// TIA Portal project "NeuroPLC_S7_1500_DB" (V21)

(* hardware
DEVICE "PLC_1"  S7-1500 station
   slot 0: "导轨_0"  Rack  6ES7 590-1***0-0AA0
   slot 1: "PLC_1"  CPU 1513-1 PN  6ES7 513-1AM03-0AB0  V3.0
      slot 3: "CPU 显示_1"  6ES7591-1AA00-0AA0
      slot 32768: "PROFINET 接口_1"  X1
         slot 32769: "端口_1"  X1 P1
         slot 32770: "端口_2"  X1 P2
      slot 34817: "Virtual CP interface port_1"  Virtual CP interface port  Virtual CP interface port
*)

// ===== PLC "PLC_1"  CPU 1513-1 PN =====

DATA_BLOCK "NeuroPLC_KAN_Weights"   // DB1
{ S7_Optimized_Access := 'TRUE' }
VERSION : 0.1
   VAR
      g0 : Array[0..49] of Real;   // LUT grid (50 pts)
      t1 : Array[0..22399] of Real;   // LUT table (16x28x50)
      w2 : Array[0..447] of Real;   // W(16x28)
      b3 : Array[0..15] of Real;   // bias(16)
      g4 : Array[0..49] of Real;   // LUT grid (50 pts)
      t5 : Array[0..3199] of Real;   // LUT table (4x16x50)
      w6 : Array[0..63] of Real;   // W(4x16)
      b7 : Array[0..3] of Real;   // bias(4)
   END_VAR
BEGIN
   g0[0] := -3.0;
   g0[1] := -2.877551;
   g0[2] := -2.755102;
   g0[3] := -2.632653;
   g0[4] := -2.510204;
   g0[5] := -2.387755;
   g0[6] := -2.265306;
   g0[7] := -2.142857;
   g0[8] := -2.020408;
   g0[9] := -1.897959;
   g0[10] := -1.77551;
   g0[11] := -1.653061;
   g0[12] := -1.530612;
   g0[13] := -1.408163;
   g0[14] := -1.285714;
   g0[15] := -1.163265;
   g0[16] := -1.040816;
   g0[17] := -0.9183673;
   g0[18] := -0.7959184;
   g0[19] := -0.6734694;
   g0[20] := -0.5510204;
   g0[21] := -0.4285714;
   g0[22] := -0.3061224;
   g0[23] := -0.1836735;
   g0[24] := -0.0612245;
   g0[25] := 0.0612245;
   g0[26] := 0.1836735;
   g0[27] := 0.3061224;
   g0[28] := 0.4285714;
   g0[29] := 0.5510204;
   g0[30] := 0.6734694;
   g0[31] := 0.7959184;
   g0[32] := 0.9183673;
   g0[33] := 1.040816;
   g0[34] := 1.163265;
   g0[35] := 1.285714;
   g0[36] := 1.408163;
   g0[37] := 1.530612;
   g0[38] := 1.653061;
   g0[39] := 1.77551;
   g0[40] := 1.897959;
   g0[41] := 2.020408;
   g0[42] := 2.142857;
   g0[43] := 2.265306;
   g0[44] := 2.387755;
   g0[45] := 2.510204;
   g0[46] := 2.632653;
   g0[47] := 2.755102;
   g0[48] := 2.877551;
   g0[49] := 3.0;
   t1[0] := -0.1194829;
   t1[1] := -0.122035;
   t1[2] := -0.1242069;
   t1[3] := -0.1259919;
   t1[4] := -0.1273833;
   t1[5] := -0.1283744;
   t1[6] := -0.1289582;
   t1[7] := -0.1291282;
   t1[8] := -0.1288773;
   t1[9] := -0.1281951;
   t1[10] := -0.1270687;
   t1[11] := -0.125485;
   t1[12] := -0.1234307;
   t1[13] := -0.120893;
   t1[14] := -0.1178586;
   t1[15] := -0.1143145;
   t1[16] := -0.1102476;
   t1[17] := -0.1056448;
   t1[18] := -0.100493;
   t1[19] := -0.0947791;
   t1[20] := -0.0884901;
   t1[21] := -0.0816128;
   t1[22] := -0.0741341;
   t1[23] := -0.066041;
   t1[24] := -0.0573203;
   t1[25] := -0.047959;
   t1[26] := -0.037944;
   t1[27] := -0.0272626;
   t1[28] := -0.0159457;
   t1[29] := -0.0041073;
   t1[30] := 0.0081295;
   t1[31] := 0.0206416;
   t1[32] := 0.033306;
   t1[33] := 0.0459995;
   t1[34] := 0.0585989;
   t1[35] := 0.0709812;
   t1[36] := 0.0830233;
   t1[37] := 0.094602;
   t1[38] := 0.1055942;
   t1[39] := 0.1158768;
   t1[40] := 0.1253268;
   t1[41] := 0.1338208;
   t1[42] := 0.141236;
   t1[43] := 0.1474491;
   t1[44] := 0.1523371;
   t1[45] := 0.1557767;
   t1[46] := 0.157645;
   t1[47] := 0.157853;
   t1[48] := 0.1564832;
   t1[49] := 0.1536715;
   t1[50] := -0.0048413;
   t1[51] := -0.005683;
   t1[52] := -0.0062711;
   t1[53] := -0.0065729;
   t1[54] := -0.0065558;
   t1[55] := -0.0061871;
   t1[56] := -0.0054341;
   t1[57] := -0.0042641;
   t1[58] := -0.0026466;
   t1[59] := -0.000584;
   t1[60] := 0.0018956;
   t1[61] := 0.0047632;
   t1[62] := 0.0079898;
   t1[63] := 0.0115464;
   t1[64] := 0.0154041;
   t1[65] := 0.0195339;
   t1[66] := 0.023907;
   t1[67] := 0.0284943;
   t1[68] := 0.0332668;
   t1[69] := 0.0381957;
   t1[70] := 0.043252;
   t1[71] := 0.0484067;
   t1[72] := 0.0536308;
   t1[73] := 0.0588955;
   t1[74] := 0.0641717;
   t1[75] := 0.0694305;
   t1[76] := 0.074643;
   t1[77] := 0.0797802;
   t1[78] := 0.0848193;
   t1[79] := 0.0897488;
   t1[80] := 0.0945588;
   t1[81] := 0.0992389;
   t1[82] := 0.1037792;
   t1[83] := 0.1081694;
   t1[84] := 0.1123995;
   t1[85] := 0.1164593;
   t1[86] := 0.1203387;
   t1[87] := 0.1240276;
   t1[88] := 0.1275157;
   t1[89] := 0.1307932;
   t1[90] := 0.1338497;
   t1[91] := 0.1366751;
   t1[92] := 0.1392594;
   t1[93] := 0.1415924;
   t1[94] := 0.143664;
   t1[95] := 0.145464;
   t1[96] := 0.1469824;
   t1[97] := 0.148212;
   t1[98] := 0.1491608;
   t1[99] := 0.1498416;
   t1[100] := -0.08693;
   t1[101] := -0.0868943;
   t1[102] := -0.0860951;
   t1[103] := -0.0844797;
   t1[104] := -0.0819952;
   t1[105] := -0.0785887;
   t1[106] := -0.0742075;
   t1[107] := -0.0687987;
   t1[108] := -0.062315;
   t1[109] := -0.054794;
   t1[110] := -0.0463402;
   t1[111] := -0.0370597;
   t1[112] := -0.027059;
   t1[113] := -0.0164442;
   t1[114] := -0.0053218;
   t1[115] := 0.0062022;
   t1[116] := 0.0180213;
   t1[117] := 0.0300293;
   t1[118] := 0.0421199;
   t1[119] := 0.0541869;
   t1[120] := 0.0661239;
   t1[121] := 0.0778248;
   t1[122] := 0.0891831;
   t1[123] := 0.1000927;
   t1[124] := 0.1104472;
   t1[125] := 0.1201404;
   t1[126] := 0.1290659;
   t1[127] := 0.137118;
   t1[128] := 0.144237;
   t1[129] := 0.1504508;
   t1[130] := 0.1557971;
   t1[131] := 0.1603135;
   t1[132] := 0.164038;
   t1[133] := 0.167008;
   t1[134] := 0.1692614;
   t1[135] := 0.1708359;
   t1[136] := 0.1717691;
   t1[137] := 0.1720988;
   t1[138] := 0.1718626;
   t1[139] := 0.1710983;
   t1[140] := 0.1698437;
   t1[141] := 0.1681363;
   t1[142] := 0.166014;
   t1[143] := 0.1635143;
   t1[144] := 0.1606752;
   t1[145] := 0.1575341;
   t1[146] := 0.1541289;
   t1[147] := 0.1504959;
   t1[148] := 0.1466652;
   t1[149] := 0.1426646;
   t1[150] := -0.0762567;
   t1[151] := -0.0788049;
   t1[152] := -0.0811656;
   t1[153] := -0.0833268;
   t1[154] := -0.0852762;
   t1[155] := -0.0870019;
   t1[156] := -0.0884917;
   t1[157] := -0.0897336;
   t1[158] := -0.0907153;
   t1[159] := -0.0914228;
   t1[160] := -0.0918409;
   t1[161] := -0.0919541;
   t1[162] := -0.0917472;
   t1[163] := -0.0912047;
   t1[164] := -0.0903113;
   t1[165] := -0.0890516;
   t1[166] := -0.0874103;
   t1[167] := -0.0853719;
   t1[168] := -0.0829212;
   t1[169] := -0.0800428;
   t1[170] := -0.0767213;
   t1[171] := -0.0729412;
   t1[172] := -0.0686874;
   t1[173] := -0.0639444;
   t1[174] := -0.0586968;
   t1[175] := -0.0529293;
   t1[176] := -0.0466265;
   t1[177] := -0.0397733;
   t1[178] := -0.0323818;
   t1[179] := -0.0245156;
   t1[180] := -0.0162441;
   t1[181] := -0.0076365;
   t1[182] := 0.0012375;
   t1[183] := 0.0103088;
   t1[184] := 0.0195079;
   t1[185] := 0.0287655;
   t1[186] := 0.0380121;
   t1[187] := 0.0471784;
   t1[188] := 0.0561951;
   t1[189] := 0.0649926;
   t1[190] := 0.0735018;
   t1[191] := 0.081653;
   t1[192] := 0.0893772;
   t1[193] := 0.0966047;
   t1[194] := 0.1032663;
   t1[195] := 0.1092926;
   t1[196] := 0.1146141;
   t1[197] := 0.1191739;
   t1[198] := 0.1229757;
   t1[199] := 0.1260427;
   t1[200] := -0.1835549;
   t1[201] := -0.1875302;
   t1[202] := -0.1909346;
   t1[203] := -0.1937087;
   t1[204] := -0.1957933;
   t1[205] := -0.1971291;
   t1[206] := -0.1976567;
   t1[207] := -0.1973169;
   t1[208] := -0.1960545;
   t1[209] := -0.1938767;
   t1[210] := -0.1908398;
   t1[211] := -0.1870016;
   t1[212] := -0.1824198;
   t1[213] := -0.1771521;
   t1[214] := -0.1712564;
   t1[215] := -0.1647903;
   t1[216] := -0.1578115;
   t1[217] := -0.1503778;
   t1[218] := -0.1425468;
   t1[219] := -0.1343765;
   t1[220] := -0.1259243;
   t1[221] := -0.1172482;
   t1[222] := -0.1084058;
   t1[223] := -0.0994548;
   t1[224] := -0.090453;
   t1[225] := -0.0814582;
   t1[226] := -0.072528;
   t1[227] := -0.0637199;
   t1[228] := -0.055075;
   t1[229] := -0.0466024;
   t1[230] := -0.0383076;
   t1[231] := -0.0301963;
   t1[232] := -0.0222742;
   t1[233] := -0.0145468;
   t1[234] := -0.0070199;
   t1[235] := 0.000301;
   t1[236] := 0.0074102;
   t1[237] := 0.0143022;
   t1[238] := 0.0209712;
   t1[239] := 0.0274116;
   t1[240] := 0.0336179;
   t1[241] := 0.0395843;
   t1[242] := 0.0453052;
   t1[243] := 0.0507751;
   t1[244] := 0.0559883;
   t1[245] := 0.0609391;
   t1[246] := 0.0656219;
   t1[247] := 0.0700293;
   t1[248] := 0.0741443;
   t1[249] := 0.077947;
   t1[250] := -0.0558672;
   t1[251] := -0.0568254;
   t1[252] := -0.0574402;
   t1[253] := -0.0577113;
   t1[254] := -0.0576384;
   t1[255] := -0.0572213;
   t1[256] := -0.0564598;
   t1[257] := -0.0553535;
   t1[258] := -0.0539027;
   t1[259] := -0.0521149;
   t1[260] := -0.0500035;
   t1[261] := -0.0475818;
   t1[262] := -0.0448633;
   t1[263] := -0.0418615;
   t1[264] := -0.0385897;
   t1[265] := -0.0350615;
   t1[266] := -0.0312902;
   t1[267] := -0.0272894;
   t1[268] := -0.0230723;
   t1[269] := -0.0186526;
   t1[270] := -0.0140436;
   t1[271] := -0.0092587;
   t1[272] := -0.0043115;
   t1[273] := 0.0007848;
   t1[274] := 0.0060165;
   t1[275] := 0.0113703;
   t1[276] := 0.0168327;
   t1[277] := 0.0223902;
   t1[278] := 0.02802;
   t1[279] := 0.0336815;
   t1[280] := 0.0393322;
   t1[281] := 0.0449295;
   t1[282] := 0.0504309;
   t1[283] := 0.0557939;
   t1[284] := 0.0609759;
   t1[285] := 0.0659345;
   t1[286] := 0.0706271;
   t1[287] := 0.0750112;
   t1[288] := 0.0790442;
   t1[289] := 0.0826836;
   t1[290] := 0.0858869;
   t1[291] := 0.0886116;
   t1[292] := 0.0908151;
   t1[293] := 0.0924549;
   t1[294] := 0.0934885;
   t1[295] := 0.0938734;
   t1[296] := 0.0935669;
   t1[297] := 0.0925394;
   t1[298] := 0.0908244;
   t1[299] := 0.0884755;
   t1[300] := 0.1269326;
   t1[301] := 0.1321426;
   t1[302] := 0.1371375;
   t1[303] := 0.1418623;
   t1[304] := 0.1462617;
   t1[305] := 0.1502807;
   t1[306] := 0.153864;
   t1[307] := 0.1569568;
   t1[308] := 0.1595052;
   t1[309] := 0.1614799;
   t1[310] := 0.1628701;
   t1[311] := 0.1636658;
   t1[312] := 0.1638568;
   t1[313] := 0.1634329;
   t1[314] := 0.1623842;
   t1[315] := 0.1607004;
   t1[316] := 0.1583713;
   t1[317] := 0.155387;
   t1[318] := 0.1517373;
   t1[319] := 0.1474119;
   t1[320] := 0.142401;
   t1[321] := 0.1366941;
   t1[322] := 0.1302814;
   t1[323] := 0.1231525;
   t1[324] := 0.1152975;
   t1[325] := 0.1067062;
   t1[326] := 0.0973684;
   t1[327] := 0.0872743;
   t1[328] := 0.0764416;
   t1[329] := 0.0649405;
   t1[330] := 0.0528468;
   t1[331] := 0.0402367;
   t1[332] := 0.0271859;
   t1[333] := 0.0137705;
   t1[334] := 6.64E-05;
   t1[335] := -0.0138503;
   t1[336] := -0.0279039;
   t1[337] := -0.0420182;
   t1[338] := -0.0561173;
   t1[339] := -0.0701254;
   t1[340] := -0.0839663;
   t1[341] := -0.0975642;
   t1[342] := -0.1108431;
   t1[343] := -0.123727;
   t1[344] := -0.1361401;
   t1[345] := -0.1480062;
   t1[346] := -0.1592495;
   t1[347] := -0.1698008;
   t1[348] := -0.1796257;
   t1[349] := -0.1887;
   t1[350] := -0.0070284;
   t1[351] := -0.0172373;
   t1[352] := -0.0269702;
   t1[353] := -0.0361019;
   t1[354] := -0.0445073;
   t1[355] := -0.0520614;
   t1[356] := -0.058639;
   t1[357] := -0.064115;
   t1[358] := -0.0683716;
   t1[359] := -0.0714012;
   t1[360] := -0.0732835;
   t1[361] := -0.0741003;
   t1[362] := -0.0739335;
   t1[363] := -0.0728651;
   t1[364] := -0.0709769;
   t1[365] := -0.0683507;
   t1[366] := -0.0650686;
   t1[367] := -0.0612124;
   t1[368] := -0.056864;
   t1[369] := -0.0521053;
   t1[370] := -0.0470183;
   t1[371] := -0.0416847;
   t1[372] := -0.0361865;
   t1[373] := -0.0306056;
   t1[374] := -0.0250239;
   t1[375] := -0.0195233;
   t1[376] := -0.0141857;
   t1[377] := -0.0090927;
   t1[378] := -0.0042989;
   t1[379] := 0.0001924;
   t1[380] := 0.0043839;
   t1[381] := 0.0082781;
   t1[382] := 0.0118774;
   t1[383] := 0.0151844;
   t1[384] := 0.0182018;
   t1[385] := 0.0209318;
   t1[386] := 0.0233773;
   t1[387] := 0.0255405;
   t1[388] := 0.0274242;
   t1[389] := 0.0290307;
   t1[390] := 0.0303627;
   t1[391] := 0.0314227;
   t1[392] := 0.0322132;
   t1[393] := 0.0327368;
   t1[394] := 0.0329959;
   t1[395] := 0.0329931;
   t1[396] := 0.032731;
   t1[397] := 0.0322134;
   t1[398] := 0.0314506;
   t1[399] := 0.0304549;
   t1[400] := -0.1028974;
   t1[401] := -0.1051299;
   t1[402] := -0.106706;
   t1[403] := -0.1075951;
   t1[404] := -0.1077664;
   t1[405] := -0.1071893;
   t1[406] := -0.1058333;
   t1[407] := -0.1036677;
   t1[408] := -0.1006654;
   t1[409] := -0.0968557;
   t1[410] := -0.0923118;
   t1[411] := -0.0871083;
   t1[412] := -0.0813197;
   t1[413] := -0.0750206;
   t1[414] := -0.0682854;
   t1[415] := -0.0611888;
   t1[416] := -0.0538051;
   t1[417] := -0.0462091;
   t1[418] := -0.0384752;
   t1[419] := -0.0306779;
   t1[420] := -0.0228918;
   t1[421] := -0.0151914;
   t1[422] := -0.0076512;
   t1[423] := -0.0003457;
   t1[424] := 0.0066504;
   t1[425] := 0.0132627;
   t1[426] := 0.0194167;
   t1[427] := 0.0250381;
   t1[428] := 0.030083;
   t1[429] := 0.0345653;
   t1[430] := 0.0385055;
   t1[431] := 0.0419237;
   t1[432] := 0.0448404;
   t1[433] := 0.0472758;
   t1[434] := 0.0492503;
   t1[435] := 0.0507842;
   t1[436] := 0.0518979;
   t1[437] := 0.0526116;
   t1[438] := 0.0529456;
   t1[439] := 0.0529204;
   t1[440] := 0.0525563;
   t1[441] := 0.0518735;
   t1[442] := 0.0508923;
   t1[443] := 0.0496332;
   t1[444] := 0.0481165;
   t1[445] := 0.0463624;
   t1[446] := 0.0443913;
   t1[447] := 0.0422223;
   t1[448] := 0.0398682;
   t1[449] := 0.0373401;
   t1[450] := 0.0462424;
   t1[451] := 0.039385;
   t1[452] := 0.0330871;
   t1[453] := 0.0274556;
   t1[454] := 0.0225975;
   t1[455] := 0.0186195;
   t1[456] := 0.0156288;
   t1[457] := 0.0137322;
   t1[458] := 0.0130303;
   t1[459] := 0.0135263;
   t1[460] := 0.0151465;
   t1[461] := 0.017815;
   t1[462] := 0.0214562;
   t1[463] := 0.0259943;
   t1[464] := 0.0313536;
   t1[465] := 0.0374582;
   t1[466] := 0.0442325;
   t1[467] := 0.0516006;
   t1[468] := 0.0594868;
   t1[469] := 0.0678154;
   t1[470] := 0.0765106;
   t1[471] := 0.0854967;
   t1[472] := 0.0946978;
   t1[473] := 0.1040383;
   t1[474] := 0.1134424;
   t1[475] := 0.1228343;
   t1[476] := 0.1321382;
   t1[477] := 0.1412786;
   t1[478] := 0.1501878;
   t1[479] := 0.1588135;
   t1[480] := 0.1671054;
   t1[481] := 0.1750129;
   t1[482] := 0.1824855;
   t1[483] := 0.1894727;
   t1[484] := 0.1959241;
   t1[485] := 0.2017891;
   t1[486] := 0.2070173;
   t1[487] := 0.2115581;
   t1[488] := 0.2153611;
   t1[489] := 0.2183758;
   t1[490] := 0.2205516;
   t1[491] := 0.2218381;
   t1[492] := 0.2221848;
   t1[493] := 0.2215413;
   t1[494] := 0.2198569;
   t1[495] := 0.2170812;
   t1[496] := 0.2131638;
   t1[497] := 0.2080761;
   t1[498] := 0.2018998;
   t1[499] := 0.1947507;
   t1[500] := 0.2054697;
   t1[501] := 0.1990182;
   t1[502] := 0.191913;
   t1[503] := 0.1842029;
   t1[504] := 0.1759365;
   t1[505] := 0.1671624;
   t1[506] := 0.1579293;
   t1[507] := 0.1482858;
   t1[508] := 0.1382816;
   t1[509] := 0.1279794;
   t1[510] := 0.1174526;
   t1[511] := 0.1067746;
   t1[512] := 0.0960191;
   t1[513] := 0.0852596;
   t1[514] := 0.0745698;
   t1[515] := 0.0640231;
   t1[516] := 0.0536932;
   t1[517] := 0.0436537;
   t1[518] := 0.0339781;
   t1[519] := 0.02474;
   t1[520] := 0.016013;
   t1[521] := 0.0078706;
   t1[522] := 0.0003865;
   t1[523] := -0.0063659;
   t1[524] := -0.0123129;
   t1[525] := -0.0173809;
   t1[526] := -0.0214963;
   t1[527] := -0.0245862;
   t1[528] := -0.0266352;
   t1[529] := -0.0277371;
   t1[530] := -0.0279982;
   t1[531] := -0.0275248;
   t1[532] := -0.0264229;
   t1[533] := -0.0247989;
   t1[534] := -0.0227588;
   t1[535] := -0.0204089;
   t1[536] := -0.0178554;
   t1[537] := -0.0152045;
   t1[538] := -0.0125623;
   t1[539] := -0.0100351;
   t1[540] := -0.007729;
   t1[541] := -0.0057503;
   t1[542] := -0.0042051;
   t1[543] := -0.0031996;
   t1[544] := -0.0028401;
   t1[545] := -0.0032327;
   t1[546] := -0.0044836;
   t1[547] := -0.0066716;
   t1[548] := -0.0097388;
   t1[549] := -0.0135843;
   t1[550] := 0.069604;
   t1[551] := 0.0578812;
   t1[552] := 0.0457085;
   t1[553] := 0.0331352;
   t1[554] := 0.0202103;
   t1[555] := 0.0069832;
   t1[556] := -0.0064972;
   t1[557] := -0.0201817;
   t1[558] := -0.0340195;
   t1[559] := -0.0479365;
   t1[560] := -0.0618403;
   t1[561] := -0.0756379;
   t1[562] := -0.0892361;
   t1[563] := -0.1025421;
   t1[564] := -0.1154626;
   t1[565] := -0.1279048;
   t1[566] := -0.1397757;
   t1[567] := -0.150982;
   t1[568] := -0.1614309;
   t1[569] := -0.1710294;
   t1[570] := -0.1796844;
   t1[571] := -0.1873028;
   t1[572] := -0.1937916;
   t1[573] := -0.1990579;
   t1[574] := -0.2030086;
   t1[575] := -0.2055506;
   t1[576] := -0.206591;
   t1[577] := -0.2060374;
   t1[578] := -0.2038705;
   t1[579] := -0.2002095;
   t1[580] := -0.1951893;
   t1[581] := -0.1889444;
   t1[582] := -0.1816098;
   t1[583] := -0.1733201;
   t1[584] := -0.16421;
   t1[585] := -0.1544143;
   t1[586] := -0.1440678;
   t1[587] := -0.1333052;
   t1[588] := -0.1222612;
   t1[589] := -0.1110705;
   t1[590] := -0.099868;
   t1[591] := -0.0887883;
   t1[592] := -0.0779662;
   t1[593] := -0.0675364;
   t1[594] := -0.0576337;
   t1[595] := -0.0483928;
   t1[596] := -0.0399484;
   t1[597] := -0.0324114;
   t1[598] := -0.0257726;
   t1[599] := -0.0199858;
   t1[600] := 0.2695681;
   t1[601] := 0.2547651;
   t1[602] := 0.2396336;
   t1[603] := 0.2242566;
   t1[604] := 0.2087173;
   t1[605] := 0.1930988;
   t1[606] := 0.177484;
   t1[607] := 0.1619561;
   t1[608] := 0.1465959;
   t1[609] := 0.1314468;
   t1[610] := 0.1165232;
   t1[611] := 0.1018386;
   t1[612] := 0.0874066;
   t1[613] := 0.0732407;
   t1[614] := 0.0593546;
   t1[615] := 0.0457617;
   t1[616] := 0.0324755;
   t1[617] := 0.0195098;
   t1[618] := 0.0068779;
   t1[619] := -0.0054066;
   t1[620] := -0.01733;
   t1[621] := -0.0288789;
   t1[622] := -0.0400397;
   t1[623] := -0.0507988;
   t1[624] := -0.0611428;
   t1[625] := -0.071058;
   t1[626] := -0.0805309;
   t1[627] := -0.089548;
   t1[628] := -0.0981051;
   t1[629] := -0.1062154;
   t1[630] := -0.1138943;
   t1[631] := -0.1211568;
   t1[632] := -0.1280182;
   t1[633] := -0.1344937;
   t1[634] := -0.1405986;
   t1[635] := -0.146348;
   t1[636] := -0.1517571;
   t1[637] := -0.1568412;
   t1[638] := -0.1616155;
   t1[639] := -0.1660953;
   t1[640] := -0.1702956;
   t1[641] := -0.1742317;
   t1[642] := -0.177919;
   t1[643] := -0.1813724;
   t1[644] := -0.1846074;
   t1[645] := -0.187639;
   t1[646] := -0.1904826;
   t1[647] := -0.1931482;
   t1[648] := -0.1956202;
   t1[649] := -0.1978753;
   t1[650] := 0.1005199;
   t1[651] := 0.1010927;
   t1[652] := 0.1019494;
   t1[653] := 0.1031047;
   t1[654] := 0.1045734;
   t1[655] := 0.1063704;
   t1[656] := 0.1085104;
   t1[657] := 0.1110083;
   t1[658] := 0.1138772;
   t1[659] := 0.1171066;
   t1[660] := 0.1206669;
   t1[661] := 0.1245281;
   t1[662] := 0.1286602;
   t1[663] := 0.1330331;
   t1[664] := 0.1376169;
   t1[665] := 0.1423814;
   t1[666] := 0.1472968;
   t1[667] := 0.1523329;
   t1[668] := 0.1574598;
   t1[669] := 0.1626474;
   t1[670] := 0.1678657;
   t1[671] := 0.1730847;
   t1[672] := 0.1782744;
   t1[673] := 0.1834047;
   t1[674] := 0.1884457;
   t1[675] := 0.1933672;
   t1[676] := 0.1981394;
   t1[677] := 0.2027322;
   t1[678] := 0.2071245;
   t1[679] := 0.2113114;
   t1[680] := 0.2152903;
   t1[681] := 0.2190582;
   t1[682] := 0.2226123;
   t1[683] := 0.2259496;
   t1[684] := 0.2290675;
   t1[685] := 0.231963;
   t1[686] := 0.2346332;
   t1[687] := 0.2370754;
   t1[688] := 0.2392866;
   t1[689] := 0.241264;
   t1[690] := 0.2430048;
   t1[691] := 0.2445061;
   t1[692] := 0.2457651;
   t1[693] := 0.2467789;
   t1[694] := 0.2475446;
   t1[695] := 0.2480595;
   t1[696] := 0.2483206;
   t1[697] := 0.2483248;
   t1[698] := 0.2480676;
   t1[699] := 0.247544;
   t1[700] := 0.0554956;
   t1[701] := 0.0394485;
   t1[702] := 0.0236316;
   t1[703] := 0.008216;
   t1[704] := -0.0066272;
   t1[705] := -0.0207266;
   t1[706] := -0.0339111;
   t1[707] := -0.0460094;
   t1[708] := -0.0568595;
   t1[709] := -0.0664407;
   t1[710] := -0.0748439;
   t1[711] := -0.0821628;
   t1[712] := -0.0884911;
   t1[713] := -0.0939227;
   t1[714] := -0.0985512;
   t1[715] := -0.1024704;
   t1[716] := -0.1057741;
   t1[717] := -0.108556;
   t1[718] := -0.1109099;
   t1[719] := -0.1129296;
   t1[720] := -0.1147089;
   t1[721] := -0.1163414;
   t1[722] := -0.1179209;
   t1[723] := -0.1195412;
   t1[724] := -0.1212961;
   t1[725] := -0.1232793;
   t1[726] := -0.1255845;
   t1[727] := -0.1283051;
   t1[728] := -0.1314804;
   t1[729] := -0.1350474;
   t1[730] := -0.1389318;
   t1[731] := -0.1430591;
   t1[732] := -0.1473549;
   t1[733] := -0.151745;
   t1[734] := -0.1561548;
   t1[735] := -0.1605101;
   t1[736] := -0.1647365;
   t1[737] := -0.1687595;
   t1[738] := -0.1725048;
   t1[739] := -0.175898;
   t1[740] := -0.1788648;
   t1[741] := -0.1813307;
   t1[742] := -0.1832213;
   t1[743] := -0.1844624;
   t1[744] := -0.1849795;
   t1[745] := -0.1846982;
   t1[746] := -0.1835442;
   t1[747] := -0.1814626;
   t1[748] := -0.178497;
   t1[749] := -0.1747214;
   t1[750] := -0.0316489;
   t1[751] := -0.0336773;
   t1[752] := -0.0356129;
   t1[753] := -0.0374797;
   t1[754] := -0.0393015;
   t1[755] := -0.0411025;
   t1[756] := -0.0429063;
   t1[757] := -0.0447371;
   t1[758] := -0.0466166;
   t1[759] := -0.0485351;
   t1[760] := -0.0504581;
   t1[761] := -0.0523502;
   t1[762] := -0.0541761;
   t1[763] := -0.0559007;
   t1[764] := -0.0574886;
   t1[765] := -0.0589045;
   t1[766] := -0.0601133;
   t1[767] := -0.0610795;
   t1[768] := -0.0617679;
   t1[769] := -0.0621433;
   t1[770] := -0.0621704;
   t1[771] := -0.0618138;
   t1[772] := -0.0610385;
   t1[773] := -0.0598089;
   t1[774] := -0.0580899;
   t1[775] := -0.0558463;
   t1[776] := -0.0530426;
   t1[777] := -0.0496441;
   t1[778] := -0.045655;
   t1[779] := -0.041154;
   t1[780] := -0.0362282;
   t1[781] := -0.0309646;
   t1[782] := -0.0254501;
   t1[783] := -0.0197719;
   t1[784] := -0.014017;
   t1[785] := -0.0082723;
   t1[786] := -0.0026249;
   t1[787] := 0.0028383;
   t1[788] := 0.00803;
   t1[789] := 0.0128635;
   t1[790] := 0.0172515;
   t1[791] := 0.0211072;
   t1[792] := 0.0243434;
   t1[793] := 0.0268733;
   t1[794] := 0.0286097;
   t1[795] := 0.0294656;
   t1[796] := 0.029354;
   t1[797] := 0.0282124;
   t1[798] := 0.0261014;
   t1[799] := 0.0231194;
   t1[800] := -0.0541978;
   t1[801] := -0.0467753;
   t1[802] := -0.0388649;
   t1[803] := -0.0305291;
   t1[804] := -0.0218303;
   t1[805] := -0.0128309;
   t1[806] := -0.0035936;
   t1[807] := 0.0058194;
   t1[808] := 0.0153467;
   t1[809] := 0.0249448;
   t1[810] := 0.0345843;
   t1[811] := 0.0442363;
   t1[812] := 0.0538718;
   t1[813] := 0.0634616;
   t1[814] := 0.0729769;
   t1[815] := 0.0823886;
   t1[816] := 0.0916676;
   t1[817] := 0.1007851;
   t1[818] := 0.1097119;
   t1[819] := 0.118419;
   t1[820] := 0.1268776;
   t1[821] := 0.1350584;
   t1[822] := 0.1429326;
   t1[823] := 0.1504711;
   t1[824] := 0.1576449;
   t1[825] := 0.164425;
   t1[826] := 0.1707824;
   t1[827] := 0.1766881;
   t1[828] := 0.1821203;
   t1[829] := 0.1870701;
   t1[830] := 0.1915307;
   t1[831] := 0.1954946;
   t1[832] := 0.1989548;
   t1[833] := 0.2019042;
   t1[834] := 0.2043355;
   t1[835] := 0.2062417;
   t1[836] := 0.2076155;
   t1[837] := 0.2084498;
   t1[838] := 0.2087374;
   t1[839] := 0.2084712;
   t1[840] := 0.2076441;
   t1[841] := 0.2062487;
   t1[842] := 0.2042782;
   t1[843] := 0.2017251;
   t1[844] := 0.1985825;
   t1[845] := 0.1948431;
   t1[846] := 0.1904997;
   t1[847] := 0.1855553;
   t1[848] := 0.1800624;
   t1[849] := 0.1740892;
   t1[850] := 0.0165106;
   t1[851] := 0.0131955;
   t1[852] := 0.0096175;
   t1[853] := 0.0058087;
   t1[854] := 0.0018013;
   t1[855] := -0.0023724;
   t1[856] := -0.0066803;
   t1[857] := -0.0110902;
   t1[858] := -0.0155693;
   t1[859] := -0.020078;
   t1[860] := -0.0245705;
   t1[861] := -0.0290012;
   t1[862] := -0.0333244;
   t1[863] := -0.0374945;
   t1[864] := -0.0414656;
   t1[865] := -0.0451922;
   t1[866] := -0.0486286;
   t1[867] := -0.051729;
   t1[868] := -0.0544477;
   t1[869] := -0.0567391;
   t1[870] := -0.0585574;
   t1[871] := -0.059857;
   t1[872] := -0.0605922;
   t1[873] := -0.0607173;
   t1[874] := -0.0601865;
   t1[875] := -0.0589543;
   t1[876] := -0.0569748;
   t1[877] := -0.0542027;
   t1[878] := -0.050625;
   t1[879] := -0.0462901;
   t1[880] := -0.0412532;
   t1[881] := -0.0355697;
   t1[882] := -0.0292946;
   t1[883] := -0.0224833;
   t1[884] := -0.0151911;
   t1[885] := -0.0074732;
   t1[886] := 0.0006152;
   t1[887] := 0.0090187;
   t1[888] := 0.0176823;
   t1[889] := 0.0265505;
   t1[890] := 0.0355681;
   t1[891] := 0.0446799;
   t1[892] := 0.0538307;
   t1[893] := 0.0629652;
   t1[894] := 0.072028;
   t1[895] := 0.0809641;
   t1[896] := 0.089718;
   t1[897] := 0.0982373;
   t1[898] := 0.1064823;
   t1[899] := 0.1144174;
   t1[900] := 0.2570028;
   t1[901] := 0.2452174;
   t1[902] := 0.2328795;
   t1[903] := 0.2200509;
   t1[904] := 0.2067933;
   t1[905] := 0.1931687;
   t1[906] := 0.1792386;
   t1[907] := 0.1650651;
   t1[908] := 0.150709;
   t1[909] := 0.1362187;
   t1[910] := 0.1216325;
   t1[911] := 0.1069886;
   t1[912] := 0.0923249;
   t1[913] := 0.0776796;
   t1[914] := 0.0630908;
   t1[915] := 0.0485965;
   t1[916] := 0.0342347;
   t1[917] := 0.0200437;
   t1[918] := 0.0060615;
   t1[919] := -0.0076739;
   t1[920] := -0.0211244;
   t1[921] := -0.0342518;
   t1[922] := -0.0470182;
   t1[923] := -0.0593854;
   t1[924] := -0.0713153;
   t1[925] := -0.0827699;
   t1[926] := -0.0937111;
   t1[927] := -0.1041009;
   t1[928] := -0.1139093;
   t1[929] := -0.1231216;
   t1[930] := -0.131725;
   t1[931] := -0.1397063;
   t1[932] := -0.1470526;
   t1[933] := -0.1537509;
   t1[934] := -0.1597883;
   t1[935] := -0.1651517;
   t1[936] := -0.1698283;
   t1[937] := -0.1738049;
   t1[938] := -0.1770687;
   t1[939] := -0.1796066;
   t1[940] := -0.1814057;
   t1[941] := -0.182453;
   t1[942] := -0.1827355;
   t1[943] := -0.1822402;
   t1[944] := -0.1809543;
   t1[945] := -0.1788645;
   t1[946] := -0.1759581;
   t1[947] := -0.172232;
   t1[948] := -0.1677332;
   t1[949] := -0.1625242;
   t1[950] := 0.1695031;
   t1[951] := 0.1635204;
   t1[952] := 0.1571902;
   t1[953] := 0.1505017;
   t1[954] := 0.1434443;
   t1[955] := 0.1360076;
   t1[956] := 0.1281809;
   t1[957] := 0.1199536;
   t1[958] := 0.1113172;
   t1[959] := 0.1022939;
   t1[960] := 0.0929304;
   t1[961] := 0.0832739;
   t1[962] := 0.0733716;
   t1[963] := 0.063271;
   t1[964] := 0.0530191;
   t1[965] := 0.0426633;
   t1[966] := 0.0322509;
   t1[967] := 0.021829;
   t1[968] := 0.0114451;
   t1[969] := 0.0011463;
   t1[970] := -0.0090201;
   t1[971] := -0.0190068;
   t1[972] := -0.0287666;
   t1[973] := -0.0382521;
   t1[974] := -0.0474162;
   t1[975] := -0.0562116;
   t1[976] := -0.0645909;
   t1[977] := -0.0725072;
   t1[978] := -0.0799368;
   t1[979] := -0.0869006;
   t1[980] := -0.0934244;
   t1[981] := -0.099534;
   t1[982] := -0.1052553;
   t1[983] := -0.1106141;
   t1[984] := -0.1156361;
   t1[985] := -0.1203473;
   t1[986] := -0.1247734;
   t1[987] := -0.1289402;
   t1[988] := -0.1328736;
   t1[989] := -0.1365994;
   t1[990] := -0.1401433;
   t1[991] := -0.1435313;
   t1[992] := -0.1467892;
   t1[993] := -0.1499427;
   t1[994] := -0.1530177;
   t1[995] := -0.1560401;
   t1[996] := -0.1590355;
   t1[997] := -0.1620217;
   t1[998] := -0.164975;
   t1[999] := -0.1678591;
   t1[1000] := -0.189392;
   t1[1001] := -0.1768052;
   t1[1002] := -0.1641579;
   t1[1003] := -0.1515508;
   t1[1004] := -0.1390849;
   t1[1005] := -0.1268609;
   t1[1006] := -0.1149796;
   t1[1007] := -0.1035419;
   t1[1008] := -0.092643;
   t1[1009] := -0.0822929;
   t1[1010] := -0.0724342;
   t1[1011] := -0.0630079;
   t1[1012] := -0.0539548;
   t1[1013] := -0.0452158;
   t1[1014] := -0.0367318;
   t1[1015] := -0.0284437;
   t1[1016] := -0.0202924;
   t1[1017] := -0.0122187;
   t1[1018] := -0.0041636;
   t1[1019] := 0.0039321;
   t1[1020] := 0.0121275;
   t1[1021] := 0.0204816;
   t1[1022] := 0.0290537;
   t1[1023] := 0.0379028;
   t1[1024] := 0.047088;
   t1[1025] := 0.0566685;
   t1[1026] := 0.0667034;
   t1[1027] := 0.0772513;
   t1[1028] := 0.0883329;
   t1[1029] := 0.0998958;
   t1[1030] := 0.1118798;
   t1[1031] := 0.1242244;
   t1[1032] := 0.1368694;
   t1[1033] := 0.1497545;
   t1[1034] := 0.1628193;
   t1[1035] := 0.1760034;
   t1[1036] := 0.1892465;
   t1[1037] := 0.2024884;
   t1[1038] := 0.2156686;
   t1[1039] := 0.2287269;
   t1[1040] := 0.2416029;
   t1[1041] := 0.2542362;
   t1[1042] := 0.2665667;
   t1[1043] := 0.2785338;
   t1[1044] := 0.2900774;
   t1[1045] := 0.301137;
   t1[1046] := 0.3116523;
   t1[1047] := 0.321566;
   t1[1048] := 0.3308358;
   t1[1049] := 0.3394241;
   t1[1050] := -0.0330082;
   t1[1051] := -0.0413051;
   t1[1052] := -0.0491068;
   t1[1053] := -0.0562725;
   t1[1054] := -0.062661;
   t1[1055] := -0.0681315;
   t1[1056] := -0.0725428;
   t1[1057] := -0.0757542;
   t1[1058] := -0.0776326;
   t1[1059] := -0.0781712;
   t1[1060] := -0.0774618;
   t1[1061] := -0.0755992;
   t1[1062] := -0.0726782;
   t1[1063] := -0.0687934;
   t1[1064] := -0.0640394;
   t1[1065] := -0.0585112;
   t1[1066] := -0.0523032;
   t1[1067] := -0.0455102;
   t1[1068] := -0.038227;
   t1[1069] := -0.0305481;
   t1[1070] := -0.0225684;
   t1[1071] := -0.0143825;
   t1[1072] := -0.0060852;
   t1[1073] := 0.002229;
   t1[1074] := 0.0104652;
   t1[1075] := 0.0185288;
   t1[1076] := 0.026325;
   t1[1077] := 0.0337595;
   t1[1078] := 0.0407725;
   t1[1079] := 0.0473696;
   t1[1080] := 0.0535637;
   t1[1081] := 0.059368;
   t1[1082] := 0.0647953;
   t1[1083] := 0.0698586;
   t1[1084] := 0.074571;
   t1[1085] := 0.0789453;
   t1[1086] := 0.0829946;
   t1[1087] := 0.0867319;
   t1[1088] := 0.0901701;
   t1[1089] := 0.0933223;
   t1[1090] := 0.0962013;
   t1[1091] := 0.0988202;
   t1[1092] := 0.101192;
   t1[1093] := 0.1033297;
   t1[1094] := 0.1052462;
   t1[1095] := 0.1069545;
   t1[1096] := 0.1084676;
   t1[1097] := 0.109796;
   t1[1098] := 0.1109382;
   t1[1099] := 0.1118888;
   t1[1100] := -0.0263191;
   t1[1101] := -0.01451;
   t1[1102] := -0.0032086;
   t1[1103] := 0.0074345;
   t1[1104] := 0.0172688;
   t1[1105] := 0.0261435;
   t1[1106] := 0.0339082;
   t1[1107] := 0.0404122;
   t1[1108] := 0.0455144;
   t1[1109] := 0.0492193;
   t1[1110] := 0.0516466;
   t1[1111] := 0.0529186;
   t1[1112] := 0.0531581;
   t1[1113] := 0.0524875;
   t1[1114] := 0.0510294;
   t1[1115] := 0.0489064;
   t1[1116] := 0.046241;
   t1[1117] := 0.0431558;
   t1[1118] := 0.0397734;
   t1[1119] := 0.0362162;
   t1[1120] := 0.0326069;
   t1[1121] := 0.0290681;
   t1[1122] := 0.0257222;
   t1[1123] := 0.0226918;
   t1[1124] := 0.0200995;
   t1[1125] := 0.0180679;
   t1[1126] := 0.0167195;
   t1[1127] := 0.0161764;
   t1[1128] := 0.0165029;
   t1[1129] := 0.0176541;
   t1[1130] := 0.019573;
   t1[1131] := 0.0222024;
   t1[1132] := 0.0254852;
   t1[1133] := 0.0293642;
   t1[1134] := 0.0337824;
   t1[1135] := 0.0386827;
   t1[1136] := 0.0440079;
   t1[1137] := 0.049701;
   t1[1138] := 0.0557048;
   t1[1139] := 0.0619621;
   t1[1140] := 0.068416;
   t1[1141] := 0.0750092;
   t1[1142] := 0.0816847;
   t1[1143] := 0.0883854;
   t1[1144] := 0.0950541;
   t1[1145] := 0.1016337;
   t1[1146] := 0.1080671;
   t1[1147] := 0.1143009;
   t1[1148] := 0.1202996;
   t1[1149] := 0.1260335;
   t1[1150] := 0.0412466;
   t1[1151] := 0.0424801;
   t1[1152] := 0.0432831;
   t1[1153] := 0.0436424;
   t1[1154] := 0.0435449;
   t1[1155] := 0.0429775;
   t1[1156] := 0.041927;
   t1[1157] := 0.0403802;
   t1[1158] := 0.0383267;
   t1[1159] := 0.0357943;
   t1[1160] := 0.0328415;
   t1[1161] := 0.0295276;
   t1[1162] := 0.0259119;
   t1[1163] := 0.0220536;
   t1[1164] := 0.018012;
   t1[1165] := 0.0138463;
   t1[1166] := 0.0096158;
   t1[1167] := 0.0053798;
   t1[1168] := 0.0011976;
   t1[1169] := -0.0028716;
   t1[1170] := -0.0067686;
   t1[1171] := -0.010434;
   t1[1172] := -0.0138085;
   t1[1173] := -0.0168331;
   t1[1174] := -0.0194482;
   t1[1175] := -0.0215948;
   t1[1176] := -0.0232134;
   t1[1177] := -0.0242452;
   t1[1178] := -0.0246632;
   t1[1179] := -0.0245009;
   t1[1180] := -0.0237986;
   t1[1181] := -0.0225969;
   t1[1182] := -0.020936;
   t1[1183] := -0.0188563;
   t1[1184] := -0.0163981;
   t1[1185] := -0.0136019;
   t1[1186] := -0.0105081;
   t1[1187] := -0.0071569;
   t1[1188] := -0.0035887;
   t1[1189] := 0.000156;
   t1[1190] := 0.004037;
   t1[1191] := 0.0080138;
   t1[1192] := 0.0120461;
   t1[1193] := 0.0160935;
   t1[1194] := 0.0201156;
   t1[1195] := 0.0240721;
   t1[1196] := 0.0279227;
   t1[1197] := 0.0316308;
   t1[1198] := 0.0351799;
   t1[1199] := 0.0385597;
   t1[1200] := 0.1668451;
   t1[1201] := 0.157337;
   t1[1202] := 0.1473946;
   t1[1203] := 0.1370998;
   t1[1204] := 0.1265343;
   t1[1205] := 0.1157796;
   t1[1206] := 0.1049176;
   t1[1207] := 0.0940298;
   t1[1208] := 0.0831964;
   t1[1209] := 0.0724736;
   t1[1210] := 0.0618986;
   t1[1211] := 0.0515082;
   t1[1212] := 0.0413391;
   t1[1213] := 0.0314279;
   t1[1214] := 0.0218116;
   t1[1215] := 0.0125267;
   t1[1216] := 0.0036101;
   t1[1217] := -0.0049014;
   t1[1218] := -0.0129713;
   t1[1219] := -0.0205627;
   t1[1220] := -0.0276389;
   t1[1221] := -0.0341632;
   t1[1222] := -0.0400987;
   t1[1223] := -0.0454088;
   t1[1224] := -0.0500568;
   t1[1225] := -0.0540058;
   t1[1226] := -0.0572192;
   t1[1227] := -0.0596604;
   t1[1228] := -0.0613163;
   t1[1229] := -0.0622176;
   t1[1230] := -0.0624005;
   t1[1231] := -0.0619007;
   t1[1232] := -0.0607542;
   t1[1233] := -0.058997;
   t1[1234] := -0.0566648;
   t1[1235] := -0.0537936;
   t1[1236] := -0.0504193;
   t1[1237] := -0.0465778;
   t1[1238] := -0.042305;
   t1[1239] := -0.0376369;
   t1[1240] := -0.0326093;
   t1[1241] := -0.0272581;
   t1[1242] := -0.0216192;
   t1[1243] := -0.0157286;
   t1[1244] := -0.0096221;
   t1[1245] := -0.0033357;
   t1[1246] := 0.0030947;
   t1[1247] := 0.0096327;
   t1[1248] := 0.016239;
   t1[1249] := 0.0228733;
   t1[1250] := -0.2291011;
   t1[1251] := -0.2228987;
   t1[1252] := -0.216103;
   t1[1253] := -0.208726;
   t1[1254] := -0.20078;
   t1[1255] := -0.1922772;
   t1[1256] := -0.1832296;
   t1[1257] := -0.1736495;
   t1[1258] := -0.1635502;
   t1[1259] := -0.1529613;
   t1[1260] := -0.1419253;
   t1[1261] := -0.1304853;
   t1[1262] := -0.1186842;
   t1[1263] := -0.1065649;
   t1[1264] := -0.0941705;
   t1[1265] := -0.0815438;
   t1[1266] := -0.0687279;
   t1[1267] := -0.0557656;
   t1[1268] := -0.0426999;
   t1[1269] := -0.0295739;
   t1[1270] := -0.0164303;
   t1[1271] := -0.0033123;
   t1[1272] := 0.0097374;
   t1[1273] := 0.0226756;
   t1[1274] := 0.0354595;
   t1[1275] := 0.0480461;
   t1[1276] := 0.0603924;
   t1[1277] := 0.0724556;
   t1[1278] := 0.0841977;
   t1[1279] := 0.0955904;
   t1[1280] := 0.1066066;
   t1[1281] := 0.1172188;
   t1[1282] := 0.1273999;
   t1[1283] := 0.1371226;
   t1[1284] := 0.1463595;
   t1[1285] := 0.1550836;
   t1[1286] := 0.1632674;
   t1[1287] := 0.1708837;
   t1[1288] := 0.1779052;
   t1[1289] := 0.1843048;
   t1[1290] := 0.1900551;
   t1[1291] := 0.1951288;
   t1[1292] := 0.1994988;
   t1[1293] := 0.2031377;
   t1[1294] := 0.2060182;
   t1[1295] := 0.2081131;
   t1[1296] := 0.2093952;
   t1[1297] := 0.209847;
   t1[1298] := 0.2095002;
   t1[1299] := 0.2084018;
   t1[1300] := 0.0971736;
   t1[1301] := 0.0893726;
   t1[1302] := 0.0816981;
   t1[1303] := 0.0742237;
   t1[1304] := 0.0670231;
   t1[1305] := 0.0601697;
   t1[1306] := 0.0537372;
   t1[1307] := 0.0477992;
   t1[1308] := 0.0424258;
   t1[1309] := 0.0376323;
   t1[1310] := 0.0333909;
   t1[1311] := 0.0296728;
   t1[1312] := 0.0264492;
   t1[1313] := 0.023691;
   t1[1314] := 0.0213695;
   t1[1315] := 0.0194558;
   t1[1316] := 0.0179209;
   t1[1317] := 0.0167361;
   t1[1318] := 0.0158723;
   t1[1319] := 0.0153008;
   t1[1320] := 0.0149927;
   t1[1321] := 0.014919;
   t1[1322] := 0.0150509;
   t1[1323] := 0.0153595;
   t1[1324] := 0.015816;
   t1[1325] := 0.0163914;
   t1[1326] := 0.0170568;
   t1[1327] := 0.0177835;
   t1[1328] := 0.0185539;
   t1[1329] := 0.0193714;
   t1[1330] := 0.0202419;
   t1[1331] := 0.0211712;
   t1[1332] := 0.0221653;
   t1[1333] := 0.0232299;
   t1[1334] := 0.0243709;
   t1[1335] := 0.0255942;
   t1[1336] := 0.0269056;
   t1[1337] := 0.028311;
   t1[1338] := 0.0298162;
   t1[1339] := 0.0314271;
   t1[1340] := 0.0331496;
   t1[1341] := 0.0349894;
   t1[1342] := 0.0369525;
   t1[1343] := 0.0390447;
   t1[1344] := 0.0412719;
   t1[1345] := 0.0436399;
   t1[1346] := 0.0461545;
   t1[1347] := 0.0488163;
   t1[1348] := 0.0515983;
   t1[1349] := 0.0544655;
   t1[1350] := 0.1530943;
   t1[1351] := 0.1526932;
   t1[1352] := 0.151513;
   t1[1353] := 0.1494604;
   t1[1354] := 0.1464418;
   t1[1355] := 0.1423638;
   t1[1356] := 0.1371326;
   t1[1357] := 0.1306549;
   t1[1358] := 0.1228458;
   t1[1359] := 0.1137522;
   t1[1360] := 0.103525;
   t1[1361] := 0.0923181;
   t1[1362] := 0.0802852;
   t1[1363] := 0.0675802;
   t1[1364] := 0.0543566;
   t1[1365] := 0.0407684;
   t1[1366] := 0.0269692;
   t1[1367] := 0.013113;
   t1[1368] := -0.0006467;
   t1[1369] := -0.014156;
   t1[1370] := -0.0272612;
   t1[1371] := -0.0398084;
   t1[1372] := -0.051644;
   t1[1373] := -0.0626141;
   t1[1374] := -0.0725651;
   t1[1375] := -0.081343;
   t1[1376] := -0.0887943;
   t1[1377] := -0.0947657;
   t1[1378] := -0.0991863;
   t1[1379] := -0.1021403;
   t1[1380] := -0.1037292;
   t1[1381] := -0.1040546;
   t1[1382] := -0.1032181;
   t1[1383] := -0.1013212;
   t1[1384] := -0.0984656;
   t1[1385] := -0.0947527;
   t1[1386] := -0.0902843;
   t1[1387] := -0.0851617;
   t1[1388] := -0.0794867;
   t1[1389] := -0.0733608;
   t1[1390] := -0.0668855;
   t1[1391] := -0.0601624;
   t1[1392] := -0.0532932;
   t1[1393] := -0.0463793;
   t1[1394] := -0.0395223;
   t1[1395] := -0.0328239;
   t1[1396] := -0.0263856;
   t1[1397] := -0.0202947;
   t1[1398] := -0.0145677;
   t1[1399] := -0.0091988;
   t1[1400] := -0.1092411;
   t1[1401] := -0.1088026;
   t1[1402] := -0.107988;
   t1[1403] := -0.1067583;
   t1[1404] := -0.1050746;
   t1[1405] := -0.1028977;
   t1[1406] := -0.1001886;
   t1[1407] := -0.0969084;
   t1[1408] := -0.0930205;
   t1[1409] := -0.0885262;
   t1[1410] := -0.0834569;
   t1[1411] := -0.0778447;
   t1[1412] := -0.0717218;
   t1[1413] := -0.0651204;
   t1[1414] := -0.0580724;
   t1[1415] := -0.0506102;
   t1[1416] := -0.0427658;
   t1[1417] := -0.0345714;
   t1[1418] := -0.0260591;
   t1[1419] := -0.017261;
   t1[1420] := -0.0082092;
   t1[1421] := 0.0010639;
   t1[1422] := 0.0105265;
   t1[1423] := 0.0201462;
   t1[1424] := 0.0298911;
   t1[1425] := 0.0397288;
   t1[1426] := 0.0496274;
   t1[1427] := 0.0595547;
   t1[1428] := 0.0694891;
   t1[1429] := 0.0794287;
   t1[1430] := 0.0893739;
   t1[1431] := 0.0993248;
   t1[1432] := 0.109282;
   t1[1433] := 0.1192455;
   t1[1434] := 0.1292159;
   t1[1435] := 0.1391932;
   t1[1436] := 0.1491779;
   t1[1437] := 0.1591703;
   t1[1438] := 0.1691706;
   t1[1439] := 0.1791793;
   t1[1440] := 0.1891965;
   t1[1441] := 0.1992225;
   t1[1442] := 0.2092578;
   t1[1443] := 0.2193026;
   t1[1444] := 0.2293572;
   t1[1445] := 0.2394219;
   t1[1446] := 0.249497;
   t1[1447] := 0.2595751;
   t1[1448] := 0.2696103;
   t1[1449] := 0.2795447;
   t1[1450] := -0.1311382;
   t1[1451] := -0.1293386;
   t1[1452] := -0.1270692;
   t1[1453] := -0.1243363;
   t1[1454] := -0.1211458;
   t1[1455] := -0.1175041;
   t1[1456] := -0.1134172;
   t1[1457] := -0.1088914;
   t1[1458] := -0.1039331;
   t1[1459] := -0.0985572;
   t1[1460] := -0.0927844;
   t1[1461] := -0.0866358;
   t1[1462] := -0.0801324;
   t1[1463] := -0.0732953;
   t1[1464] := -0.0661454;
   t1[1465] := -0.0587038;
   t1[1466] := -0.0509916;
   t1[1467] := -0.0430297;
   t1[1468] := -0.0348392;
   t1[1469] := -0.0264412;
   t1[1470] := -0.0178567;
   t1[1471] := -0.0091066;
   t1[1472] := -0.0002121;
   t1[1473] := 0.0088059;
   t1[1474] := 0.0179262;
   t1[1475] := 0.0271279;
   t1[1476] := 0.03639;
   t1[1477] := 0.0456913;
   t1[1478] := 0.0550137;
   t1[1479] := 0.0643438;
   t1[1480] := 0.073669;
   t1[1481] := 0.0829765;
   t1[1482] := 0.0922537;
   t1[1483] := 0.1014878;
   t1[1484] := 0.1106663;
   t1[1485] := 0.1197764;
   t1[1486] := 0.1288054;
   t1[1487] := 0.1377407;
   t1[1488] := 0.1465695;
   t1[1489] := 0.1552792;
   t1[1490] := 0.163857;
   t1[1491] := 0.1722903;
   t1[1492] := 0.1805664;
   t1[1493] := 0.1886727;
   t1[1494] := 0.1965963;
   t1[1495] := 0.2043247;
   t1[1496] := 0.2118451;
   t1[1497] := 0.2191418;
   t1[1498] := 0.2261835;
   t1[1499] := 0.232934;
   t1[1500] := -0.2517078;
   t1[1501] := -0.255779;
   t1[1502] := -0.2592178;
   t1[1503] := -0.2619836;
   t1[1504] := -0.2640356;
   t1[1505] := -0.2653331;
   t1[1506] := -0.2658352;
   t1[1507] := -0.2655013;
   t1[1508] := -0.2642928;
   t1[1509] := -0.2622057;
   t1[1510] := -0.2592635;
   t1[1511] := -0.2554899;
   t1[1512] := -0.2509092;
   t1[1513] := -0.2455452;
   t1[1514] := -0.2394219;
   t1[1515] := -0.2325635;
   t1[1516] := -0.2249937;
   t1[1517] := -0.2167368;
   t1[1518] := -0.2078166;
   t1[1519] := -0.1982572;
   t1[1520] := -0.1880826;
   t1[1521] := -0.1773168;
   t1[1522] := -0.1659838;
   t1[1523] := -0.1541075;
   t1[1524] := -0.141712;
   t1[1525] := -0.1288214;
   t1[1526] := -0.1154595;
   t1[1527] := -0.1016505;
   t1[1528] := -0.0874226;
   t1[1529] := -0.0728122;
   t1[1530] := -0.0578567;
   t1[1531] := -0.0425932;
   t1[1532] := -0.0270591;
   t1[1533] := -0.0112917;
   t1[1534] := 0.0046719;
   t1[1535] := 0.0207941;
   t1[1536] := 0.0370379;
   t1[1537] := 0.0533659;
   t1[1538] := 0.0697409;
   t1[1539] := 0.0861255;
   t1[1540] := 0.1024824;
   t1[1541] := 0.1187744;
   t1[1542] := 0.1349643;
   t1[1543] := 0.1510147;
   t1[1544] := 0.1668883;
   t1[1545] := 0.1825478;
   t1[1546] := 0.197956;
   t1[1547] := 0.2130717;
   t1[1548] := 0.2278336;
   t1[1549] := 0.2421744;
   t1[1550] := 0.0492069;
   t1[1551] := 0.0473487;
   t1[1552] := 0.0448848;
   t1[1553] := 0.0417536;
   t1[1554] := 0.0378936;
   t1[1555] := 0.0332431;
   t1[1556] := 0.0277405;
   t1[1557] := 0.0213245;
   t1[1558] := 0.0139391;
   t1[1559] := 0.005619;
   t1[1560] := -0.0035302;
   t1[1561] := -0.013401;
   t1[1562] := -0.023886;
   t1[1563] := -0.0348776;
   t1[1564] := -0.0462682;
   t1[1565] := -0.0579503;
   t1[1566] := -0.0698166;
   t1[1567] := -0.0817592;
   t1[1568] := -0.0936709;
   t1[1569] := -0.1054441;
   t1[1570] := -0.1169712;
   t1[1571] := -0.1281447;
   t1[1572] := -0.1388571;
   t1[1573] := -0.149001;
   t1[1574] := -0.1584687;
   t1[1575] := -0.1671527;
   t1[1576] := -0.1749456;
   t1[1577] := -0.1817403;
   t1[1578] := -0.187479;
   t1[1579] := -0.1921975;
   t1[1580] := -0.1959424;
   t1[1581] := -0.1987597;
   t1[1582] := -0.2006959;
   t1[1583] := -0.2017973;
   t1[1584] := -0.2021101;
   t1[1585] := -0.2016807;
   t1[1586] := -0.2005555;
   t1[1587] := -0.1987807;
   t1[1588] := -0.1964026;
   t1[1589] := -0.1934676;
   t1[1590] := -0.1900219;
   t1[1591] := -0.1861119;
   t1[1592] := -0.181784;
   t1[1593] := -0.1770843;
   t1[1594] := -0.1720593;
   t1[1595] := -0.1667552;
   t1[1596] := -0.1612183;
   t1[1597] := -0.1554927;
   t1[1598] := -0.1496101;
   t1[1599] := -0.1435986;
   t1[1600] := 0.2468299;
   t1[1601] := 0.2540316;
   t1[1602] := 0.2604414;
   t1[1603] := 0.2659326;
   t1[1604] := 0.2703789;
   t1[1605] := 0.2736538;
   t1[1606] := 0.2756305;
   t1[1607] := 0.2761828;
   t1[1608] := 0.2751915;
   t1[1609] := 0.2726526;
   t1[1610] := 0.2686527;
   t1[1611] := 0.2632808;
   t1[1612] := 0.2566258;
   t1[1613] := 0.2487768;
   t1[1614] := 0.2398228;
   t1[1615] := 0.2298528;
   t1[1616] := 0.2189557;
   t1[1617] := 0.2072205;
   t1[1618] := 0.1947364;
   t1[1619] := 0.1815922;
   t1[1620] := 0.167877;
   t1[1621] := 0.1536797;
   t1[1622] := 0.1390895;
   t1[1623] := 0.1241952;
   t1[1624] := 0.1090858;
   t1[1625] := 0.0938504;
   t1[1626] := 0.078578;
   t1[1627] := 0.0633574;
   t1[1628] := 0.0482628;
   t1[1629] := 0.0333406;
   t1[1630] := 0.018634;
   t1[1631] := 0.0041861;
   t1[1632] := -0.0099597;
   t1[1633] := -0.0237602;
   t1[1634] := -0.0371722;
   t1[1635] := -0.0501526;
   t1[1636] := -0.0626579;
   t1[1637] := -0.0746451;
   t1[1638] := -0.0860709;
   t1[1639] := -0.096892;
   t1[1640] := -0.1070653;
   t1[1641] := -0.1165475;
   t1[1642] := -0.1252953;
   t1[1643] := -0.1332657;
   t1[1644] := -0.1404152;
   t1[1645] := -0.1467007;
   t1[1646] := -0.152079;
   t1[1647] := -0.1565153;
   t1[1648] := -0.1600175;
   t1[1649] := -0.1626064;
   t1[1650] := -0.0399078;
   t1[1651] := -0.0301289;
   t1[1652] := -0.0201678;
   t1[1653] := -0.0101244;
   t1[1654] := -9.84E-05;
   t1[1655] := 0.0098103;
   t1[1656] := 0.0195017;
   t1[1657] := 0.0288762;
   t1[1658] := 0.0378364;
   t1[1659] := 0.0463278;
   t1[1660] := 0.0543289;
   t1[1661] := 0.0618192;
   t1[1662] := 0.0687783;
   t1[1663] := 0.0751856;
   t1[1664] := 0.0810207;
   t1[1665] := 0.0862631;
   t1[1666] := 0.0908924;
   t1[1667] := 0.0948879;
   t1[1668] := 0.0982293;
   t1[1669] := 0.1008961;
   t1[1670] := 0.1028678;
   t1[1671] := 0.1041238;
   t1[1672] := 0.1046438;
   t1[1673] := 0.1044072;
   t1[1674] := 0.1033935;
   t1[1675] := 0.1015823;
   t1[1676] := 0.0989531;
   t1[1677] := 0.0954857;
   t1[1678] := 0.0911945;
   t1[1679] := 0.0861596;
   t1[1680] := 0.0804685;
   t1[1681] := 0.0742084;
   t1[1682] := 0.0674668;
   t1[1683] := 0.0603311;
   t1[1684] := 0.0528886;
   t1[1685] := 0.0452268;
   t1[1686] := 0.0374331;
   t1[1687] := 0.0295947;
   t1[1688] := 0.0217992;
   t1[1689] := 0.014134;
   t1[1690] := 0.0066863;
   t1[1691] := -0.0004563;
   t1[1692] := -0.0072066;
   t1[1693] := -0.0134771;
   t1[1694] := -0.0191804;
   t1[1695] := -0.0242291;
   t1[1696] := -0.0285359;
   t1[1697] := -0.0320332;
   t1[1698] := -0.0347523;
   t1[1699] := -0.0367556;
   t1[1700] := -0.227583;
   t1[1701] := -0.2247074;
   t1[1702] := -0.2216533;
   t1[1703] := -0.2184904;
   t1[1704] := -0.215288;
   t1[1705] := -0.2121158;
   t1[1706] := -0.2090431;
   t1[1707] := -0.2061395;
   t1[1708] := -0.2034693;
   t1[1709] := -0.201016;
   t1[1710] := -0.1986995;
   t1[1711] := -0.1964381;
   t1[1712] := -0.19415;
   t1[1713] := -0.1917534;
   t1[1714] := -0.1891667;
   t1[1715] := -0.186308;
   t1[1716] := -0.1830956;
   t1[1717] := -0.1794477;
   t1[1718] := -0.1752826;
   t1[1719] := -0.1705185;
   t1[1720] := -0.1650736;
   t1[1721] := -0.1588662;
   t1[1722] := -0.1518145;
   t1[1723] := -0.1438368;
   t1[1724] := -0.1348513;
   t1[1725] := -0.1247762;
   t1[1726] := -0.1135298;
   t1[1727] := -0.1010309;
   t1[1728] := -0.0872722;
   t1[1729] := -0.0723857;
   t1[1730] := -0.056519;
   t1[1731] := -0.0398198;
   t1[1732] := -0.0224358;
   t1[1733] := -0.0045147;
   t1[1734] := 0.013796;
   t1[1735] := 0.0323485;
   t1[1736] := 0.0509951;
   t1[1737] := 0.0695881;
   t1[1738] := 0.08798;
   t1[1739] := 0.1060231;
   t1[1740] := 0.1235696;
   t1[1741] := 0.140472;
   t1[1742] := 0.1565824;
   t1[1743] := 0.1717535;
   t1[1744] := 0.1858373;
   t1[1745] := 0.1986862;
   t1[1746] := 0.2101526;
   t1[1747] := 0.220115;
   t1[1748] := 0.2285822;
   t1[1749] := 0.235604;
   t1[1750] := 0.15399;
   t1[1751] := 0.1538572;
   t1[1752] := 0.1530664;
   t1[1753] := 0.1515775;
   t1[1754] := 0.1493506;
   t1[1755] := 0.1463457;
   t1[1756] := 0.1425229;
   t1[1757] := 0.1378421;
   t1[1758] := 0.1322681;
   t1[1759] := 0.1258384;
   t1[1760] := 0.1186478;
   t1[1761] := 0.1107924;
   t1[1762] := 0.1023686;
   t1[1763] := 0.0934728;
   t1[1764] := 0.084201;
   t1[1765] := 0.0746497;
   t1[1766] := 0.0649152;
   t1[1767] := 0.0550936;
   t1[1768] := 0.0452813;
   t1[1769] := 0.0355746;
   t1[1770] := 0.0260698;
   t1[1771] := 0.0168631;
   t1[1772] := 0.0080508;
   t1[1773] := -0.0002708;
   t1[1774] := -0.0080054;
   t1[1775] := -0.0150567;
   t1[1776] := -0.0213285;
   t1[1777] := -0.0267247;
   t1[1778] := -0.0311856;
   t1[1779] := -0.03472;
   t1[1780] := -0.0373441;
   t1[1781] := -0.0390743;
   t1[1782] := -0.0399271;
   t1[1783] := -0.0399188;
   t1[1784] := -0.0390658;
   t1[1785] := -0.0373845;
   t1[1786] := -0.0348912;
   t1[1787] := -0.0316023;
   t1[1788] := -0.0275342;
   t1[1789] := -0.0227033;
   t1[1790] := -0.017126;
   t1[1791] := -0.0108185;
   t1[1792] := -0.0037974;
   t1[1793] := 0.003921;
   t1[1794] := 0.0123203;
   t1[1795] := 0.0213842;
   t1[1796] := 0.0310963;
   t1[1797] := 0.0414288;
   t1[1798] := 0.0522972;
   t1[1799] := 0.063599;
   t1[1800] := -0.1692545;
   t1[1801] := -0.1719219;
   t1[1802] := -0.1737095;
   t1[1803] := -0.1745087;
   t1[1804] := -0.1742106;
   t1[1805] := -0.1727067;
   t1[1806] := -0.1698882;
   t1[1807] := -0.1656465;
   t1[1808] := -0.1598818;
   t1[1809] := -0.1526316;
   t1[1810] := -0.1440417;
   t1[1811] := -0.1342608;
   t1[1812] := -0.1234376;
   t1[1813] := -0.1117208;
   t1[1814] := -0.099259;
   t1[1815] := -0.086201;
   t1[1816] := -0.0726953;
   t1[1817] := -0.0588908;
   t1[1818] := -0.044936;
   t1[1819] := -0.0309797;
   t1[1820] := -0.0171706;
   t1[1821] := -0.0036572;
   t1[1822] := 0.0094116;
   t1[1823] := 0.0218873;
   t1[1824] := 0.0336211;
   t1[1825] := 0.0444643;
   t1[1826] := 0.0542682;
   t1[1827] := 0.062885;
   t1[1828] := 0.0702438;
   t1[1829] := 0.0764204;
   t1[1830] := 0.0815068;
   t1[1831] := 0.0855952;
   t1[1832] := 0.0887777;
   t1[1833] := 0.0911463;
   t1[1834] := 0.092793;
   t1[1835] := 0.0938102;
   t1[1836] := 0.0942897;
   t1[1837] := 0.0943237;
   t1[1838] := 0.0940042;
   t1[1839] := 0.0934234;
   t1[1840] := 0.0926734;
   t1[1841] := 0.0918462;
   t1[1842] := 0.091034;
   t1[1843] := 0.0903287;
   t1[1844] := 0.0898226;
   t1[1845] := 0.0896076;
   t1[1846] := 0.089776;
   t1[1847] := 0.090402;
   t1[1848] := 0.0914717;
   t1[1849] := 0.0929436;
   t1[1850] := -0.1842585;
   t1[1851] := -0.1840431;
   t1[1852] := -0.1834812;
   t1[1853] := -0.1824941;
   t1[1854] := -0.1810031;
   t1[1855] := -0.1789295;
   t1[1856] := -0.1761944;
   t1[1857] := -0.1727193;
   t1[1858] := -0.1684293;
   t1[1859] := -0.1633116;
   t1[1860] := -0.1574021;
   t1[1861] := -0.1507379;
   t1[1862] := -0.1433562;
   t1[1863] := -0.1352942;
   t1[1864] := -0.126589;
   t1[1865] := -0.1172778;
   t1[1866] := -0.1073979;
   t1[1867] := -0.0969863;
   t1[1868] := -0.0860802;
   t1[1869] := -0.0747169;
   t1[1870] := -0.0629335;
   t1[1871] := -0.050767;
   t1[1872] := -0.0382549;
   t1[1873] := -0.0254341;
   t1[1874] := -0.0123419;
   t1[1875] := 0.0009846;
   t1[1876] := 0.0145081;
   t1[1877] := 0.0281916;
   t1[1878] := 0.0420004;
   t1[1879] := 0.0559045;
   t1[1880] := 0.0698747;
   t1[1881] := 0.0838816;
   t1[1882] := 0.0978958;
   t1[1883] := 0.1118879;
   t1[1884] := 0.1258287;
   t1[1885] := 0.1396887;
   t1[1886] := 0.1534386;
   t1[1887] := 0.167049;
   t1[1888] := 0.1804906;
   t1[1889] := 0.1937339;
   t1[1890] := 0.2067497;
   t1[1891] := 0.2195086;
   t1[1892] := 0.2319812;
   t1[1893] := 0.2441382;
   t1[1894] := 0.2559501;
   t1[1895] := 0.2673877;
   t1[1896] := 0.2784216;
   t1[1897] := 0.2890209;
   t1[1898] := 0.2991468;
   t1[1899] := 0.3087583;
   t1[1900] := -0.3433722;
   t1[1901] := -0.3352931;
   t1[1902] := -0.3264073;
   t1[1903] := -0.3167214;
   t1[1904] := -0.3062419;
   t1[1905] := -0.2949751;
   t1[1906] := -0.2829276;
   t1[1907] := -0.2701057;
   t1[1908] := -0.2565185;
   t1[1909] := -0.2422126;
   t1[1910] := -0.2272647;
   t1[1911] := -0.2117521;
   t1[1912] := -0.1957523;
   t1[1913] := -0.1793427;
   t1[1914] := -0.1626008;
   t1[1915] := -0.1456038;
   t1[1916] := -0.1284292;
   t1[1917] := -0.1111544;
   t1[1918] := -0.0938568;
   t1[1919] := -0.0766139;
   t1[1920] := -0.059503;
   t1[1921] := -0.0426015;
   t1[1922] := -0.0259869;
   t1[1923] := -0.0097365;
   t1[1924] := 0.0060723;
   t1[1925] := 0.021362;
   t1[1926] := 0.0360552;
   t1[1927] := 0.0500748;
   t1[1928] := 0.0633724;
   t1[1929] := 0.0759543;
   t1[1930] := 0.0878328;
   t1[1931] := 0.0990201;
   t1[1932] := 0.1095287;
   t1[1933] := 0.1193707;
   t1[1934] := 0.1285587;
   t1[1935] := 0.1371047;
   t1[1936] := 0.1450212;
   t1[1937] := 0.1523206;
   t1[1938] := 0.159015;
   t1[1939] := 0.1651168;
   t1[1940] := 0.1706384;
   t1[1941] := 0.175592;
   t1[1942] := 0.17999;
   t1[1943] := 0.1838447;
   t1[1944] := 0.1871684;
   t1[1945] := 0.1899734;
   t1[1946] := 0.192272;
   t1[1947] := 0.1940764;
   t1[1948] := 0.1953979;
   t1[1949] := 0.1962473;
   t1[1950] := 0.0363517;
   t1[1951] := 0.0309942;
   t1[1952] := 0.0259224;
   t1[1953] := 0.0212328;
   t1[1954] := 0.0170217;
   t1[1955] := 0.0133855;
   t1[1956] := 0.0104207;
   t1[1957] := 0.0082236;
   t1[1958] := 0.0068848;
   t1[1959] := 0.0064029;
   t1[1960] := 0.0067043;
   t1[1961] := 0.0077135;
   t1[1962] := 0.0093549;
   t1[1963] := 0.0115529;
   t1[1964] := 0.0142321;
   t1[1965] := 0.0173167;
   t1[1966] := 0.0207314;
   t1[1967] := 0.0244004;
   t1[1968] := 0.0282484;
   t1[1969] := 0.0321997;
   t1[1970] := 0.0361787;
   t1[1971] := 0.0401099;
   t1[1972] := 0.0439178;
   t1[1973] := 0.0475268;
   t1[1974] := 0.0508614;
   t1[1975] := 0.0538459;
   t1[1976] := 0.0564049;
   t1[1977] := 0.058463;
   t1[1978] := 0.059982;
   t1[1979] := 0.0609932;
   t1[1980] := 0.0615358;
   t1[1981] := 0.0616491;
   t1[1982] := 0.0613721;
   t1[1983] := 0.0607442;
   t1[1984] := 0.0598046;
   t1[1985] := 0.0585923;
   t1[1986] := 0.0571468;
   t1[1987] := 0.055507;
   t1[1988] := 0.0537123;
   t1[1989] := 0.0518019;
   t1[1990] := 0.0498149;
   t1[1991] := 0.0477906;
   t1[1992] := 0.0457681;
   t1[1993] := 0.0437867;
   t1[1994] := 0.0418856;
   t1[1995] := 0.040104;
   t1[1996] := 0.038481;
   t1[1997] := 0.0370488;
   t1[1998] := 0.0358042;
   t1[1999] := 0.0347328;
   t1[2000] := -0.2135215;
   t1[2001] := -0.1983883;
   t1[2002] := -0.1827447;
   t1[2003] := -0.166669;
   t1[2004] := -0.1502396;
   t1[2005] := -0.1335349;
   t1[2006] := -0.1166332;
   t1[2007] := -0.0996131;
   t1[2008] := -0.0825521;
   t1[2009] := -0.0655172;
   t1[2010] := -0.0485664;
   t1[2011] := -0.0317578;
   t1[2012] := -0.0151492;
   t1[2013] := 0.0012013;
   t1[2014] := 0.0172358;
   t1[2015] := 0.0328962;
   t1[2016] := 0.0481248;
   t1[2017] := 0.0628634;
   t1[2018] := 0.0770541;
   t1[2019] := 0.090639;
   t1[2020] := 0.1035601;
   t1[2021] := 0.1157594;
   t1[2022] := 0.127179;
   t1[2023] := 0.1377609;
   t1[2024] := 0.1474471;
   t1[2025] := 0.1561797;
   t1[2026] := 0.1639007;
   t1[2027] := 0.1705526;
   t1[2028] := 0.1761245;
   t1[2029] := 0.1806938;
   t1[2030] := 0.1843482;
   t1[2031] := 0.1871748;
   t1[2032] := 0.1892613;
   t1[2033] := 0.190695;
   t1[2034] := 0.1915633;
   t1[2035] := 0.1919536;
   t1[2036] := 0.1919534;
   t1[2037] := 0.1916501;
   t1[2038] := 0.1911311;
   t1[2039] := 0.1904838;
   t1[2040] := 0.1897957;
   t1[2041] := 0.1891541;
   t1[2042] := 0.1886465;
   t1[2043] := 0.1883604;
   t1[2044] := 0.188383;
   t1[2045] := 0.1888019;
   t1[2046] := 0.1897045;
   t1[2047] := 0.191155;
   t1[2048] := 0.1931011;
   t1[2049] := 0.1954547;
   t1[2050] := -0.2638247;
   t1[2051] := -0.253926;
   t1[2052] := -0.243357;
   t1[2053] := -0.232141;
   t1[2054] := -0.2203012;
   t1[2055] := -0.2078611;
   t1[2056] := -0.1948439;
   t1[2057] := -0.181273;
   t1[2058] := -0.167174;
   t1[2059] := -0.1526075;
   t1[2060] := -0.1376618;
   t1[2061] := -0.1224262;
   t1[2062] := -0.1069895;
   t1[2063] := -0.0914409;
   t1[2064] := -0.0758695;
   t1[2065] := -0.0603644;
   t1[2066] := -0.0450145;
   t1[2067] := -0.0299091;
   t1[2068] := -0.0151371;
   t1[2069] := -0.0007877;
   t1[2070] := 0.0130502;
   t1[2071] := 0.0262873;
   t1[2072] := 0.0388347;
   t1[2073] := 0.0506033;
   t1[2074] := 0.061504;
   t1[2075] := 0.0714477;
   t1[2076] := 0.0803453;
   t1[2077] := 0.0881083;
   t1[2078] := 0.0947028;
   t1[2079] := 0.1001986;
   t1[2080] := 0.104677;
   t1[2081] := 0.1082193;
   t1[2082] := 0.1109071;
   t1[2083] := 0.1128215;
   t1[2084] := 0.114044;
   t1[2085] := 0.114656;
   t1[2086] := 0.1147388;
   t1[2087] := 0.1143738;
   t1[2088] := 0.1136424;
   t1[2089] := 0.1126258;
   t1[2090] := 0.1114055;
   t1[2091] := 0.1100629;
   t1[2092] := 0.1086792;
   t1[2093] := 0.1073359;
   t1[2094] := 0.1061144;
   t1[2095] := 0.1050959;
   t1[2096] := 0.1043619;
   t1[2097] := 0.1039764;
   t1[2098] := 0.1039163;
   t1[2099] := 0.1041317;
   t1[2100] := -0.0215827;
   t1[2101] := -0.0217664;
   t1[2102] := -0.0220519;
   t1[2103] := -0.0223617;
   t1[2104] := -0.0226185;
   t1[2105] := -0.0227447;
   t1[2106] := -0.0226629;
   t1[2107] := -0.0222959;
   t1[2108] := -0.0215713;
   t1[2109] := -0.0204994;
   t1[2110] := -0.0191547;
   t1[2111] := -0.0176138;
   t1[2112] := -0.015953;
   t1[2113] := -0.0142488;
   t1[2114] := -0.0125777;
   t1[2115] := -0.0110161;
   t1[2116] := -0.0096404;
   t1[2117] := -0.0085271;
   t1[2118] := -0.0077527;
   t1[2119] := -0.0073935;
   t1[2120] := -0.007526;
   t1[2121] := -0.0082266;
   t1[2122] := -0.0095719;
   t1[2123] := -0.0116382;
   t1[2124] := -0.014502;
   t1[2125] := -0.0182397;
   t1[2126] := -0.0229278;
   t1[2127] := -0.0286421;
   t1[2128] := -0.0353979;
   t1[2129] := -0.0430952;
   t1[2130] := -0.0516213;
   t1[2131] := -0.0608633;
   t1[2132] := -0.0707085;
   t1[2133] := -0.081044;
   t1[2134] := -0.0917572;
   t1[2135] := -0.1027351;
   t1[2136] := -0.1138651;
   t1[2137] := -0.1250344;
   t1[2138] := -0.1361301;
   t1[2139] := -0.1470395;
   t1[2140] := -0.1576497;
   t1[2141] := -0.1678481;
   t1[2142] := -0.1775218;
   t1[2143] := -0.1865581;
   t1[2144] := -0.1948441;
   t1[2145] := -0.202267;
   t1[2146] := -0.2087142;
   t1[2147] := -0.2140943;
   t1[2148] := -0.2184236;
   t1[2149] := -0.2217521;
   t1[2150] := 0.0948695;
   t1[2151] := 0.1027036;
   t1[2152] := 0.1098262;
   t1[2153] := 0.116154;
   t1[2154] := 0.1216037;
   t1[2155] := 0.1260919;
   t1[2156] := 0.1295351;
   t1[2157] := 0.1318502;
   t1[2158] := 0.1329586;
   t1[2159] := 0.132856;
   t1[2160] := 0.131597;
   t1[2161] := 0.1292376;
   t1[2162] := 0.1258339;
   t1[2163] := 0.1214417;
   t1[2164] := 0.1161173;
   t1[2165] := 0.1099166;
   t1[2166] := 0.1028956;
   t1[2167] := 0.0951103;
   t1[2168] := 0.0866169;
   t1[2169] := 0.0774713;
   t1[2170] := 0.0677295;
   t1[2171] := 0.0574476;
   t1[2172] := 0.0466816;
   t1[2173] := 0.0354875;
   t1[2174] := 0.0239214;
   t1[2175] := 0.0120393;
   t1[2176] := -0.0001028;
   t1[2177] := -0.0124489;
   t1[2178] := -0.0249446;
   t1[2179] := -0.0375386;
   t1[2180] := -0.05018;
   t1[2181] := -0.0628179;
   t1[2182] := -0.0754015;
   t1[2183] := -0.0878796;
   t1[2184] := -0.1002016;
   t1[2185] := -0.1123164;
   t1[2186] := -0.1241731;
   t1[2187] := -0.1357209;
   t1[2188] := -0.1469087;
   t1[2189] := -0.1576857;
   t1[2190] := -0.168001;
   t1[2191] := -0.1778036;
   t1[2192] := -0.1870427;
   t1[2193] := -0.1956673;
   t1[2194] := -0.2036265;
   t1[2195] := -0.2108694;
   t1[2196] := -0.217345;
   t1[2197] := -0.2230122;
   t1[2198] := -0.2278775;
   t1[2199] := -0.2319627;
   t1[2200] := 0.2239106;
   t1[2201] := 0.2190618;
   t1[2202] := 0.2131876;
   t1[2203] := 0.2063059;
   t1[2204] := 0.1984346;
   t1[2205] := 0.1895914;
   t1[2206] := 0.1797942;
   t1[2207] := 0.1690608;
   t1[2208] := 0.1574113;
   t1[2209] := 0.144899;
   t1[2210] := 0.1316038;
   t1[2211] := 0.1176062;
   t1[2212] := 0.1029866;
   t1[2213] := 0.0878256;
   t1[2214] := 0.0722037;
   t1[2215] := 0.0562014;
   t1[2216] := 0.0398991;
   t1[2217] := 0.0233774;
   t1[2218] := 0.0067168;
   t1[2219] := -0.0100023;
   t1[2220] := -0.0266993;
   t1[2221] := -0.0432937;
   t1[2222] := -0.059705;
   t1[2223] := -0.0758528;
   t1[2224] := -0.0916565;
   t1[2225] := -0.1070356;
   t1[2226] := -0.1219096;
   t1[2227] := -0.1361983;
   t1[2228] := -0.1498503;
   t1[2229] := -0.1628686;
   t1[2230] := -0.1752626;
   t1[2231] := -0.1870415;
   t1[2232] := -0.1982146;
   t1[2233] := -0.208791;
   t1[2234] := -0.2187801;
   t1[2235] := -0.228191;
   t1[2236] := -0.2370331;
   t1[2237] := -0.2453157;
   t1[2238] := -0.2530478;
   t1[2239] := -0.2602389;
   t1[2240] := -0.2668981;
   t1[2241] := -0.2730347;
   t1[2242] := -0.278658;
   t1[2243] := -0.2837772;
   t1[2244] := -0.2884016;
   t1[2245] := -0.2925403;
   t1[2246] := -0.2962027;
   t1[2247] := -0.2993954;
   t1[2248] := -0.3021117;
   t1[2249] := -0.3043406;
   t1[2250] := -0.210152;
   t1[2251] := -0.1990302;
   t1[2252] := -0.1876812;
   t1[2253] := -0.1762033;
   t1[2254] := -0.1646952;
   t1[2255] := -0.153255;
   t1[2256] := -0.1419814;
   t1[2257] := -0.1309727;
   t1[2258] := -0.1203236;
   t1[2259] := -0.1100722;
   t1[2260] := -0.1002113;
   t1[2261] := -0.0907329;
   t1[2262] := -0.0816288;
   t1[2263] := -0.072891;
   t1[2264] := -0.0645113;
   t1[2265] := -0.0564815;
   t1[2266] := -0.0487936;
   t1[2267] := -0.0414393;
   t1[2268] := -0.0344107;
   t1[2269] := -0.0276995;
   t1[2270] := -0.0212975;
   t1[2271] := -0.0151968;
   t1[2272] := -0.0093891;
   t1[2273] := -0.0038663;
   t1[2274] := 0.0013797;
   t1[2275] := 0.006357;
   t1[2276] := 0.0110738;
   t1[2277] := 0.0155381;
   t1[2278] := 0.0197446;
   t1[2279] := 0.0236629;
   t1[2280] := 0.0272598;
   t1[2281] := 0.030502;
   t1[2282] := 0.0333564;
   t1[2283] := 0.0357896;
   t1[2284] := 0.0377684;
   t1[2285] := 0.0392597;
   t1[2286] := 0.0402302;
   t1[2287] := 0.0406466;
   t1[2288] := 0.0404757;
   t1[2289] := 0.0396844;
   t1[2290] := 0.0382393;
   t1[2291] := 0.0361072;
   t1[2292] := 0.0332549;
   t1[2293] := 0.0296492;
   t1[2294] := 0.0252568;
   t1[2295] := 0.0200445;
   t1[2296] := 0.0139791;
   t1[2297] := 0.0070468;
   t1[2298] := -0.000669;
   t1[2299] := -0.0090543;
   t1[2300] := -0.2450845;
   t1[2301] := -0.2353242;
   t1[2302] := -0.2247794;
   t1[2303] := -0.2134059;
   t1[2304] := -0.2011592;
   t1[2305] := -0.1879949;
   t1[2306] := -0.1738686;
   t1[2307] := -0.1587359;
   t1[2308] := -0.1425592;
   t1[2309] := -0.1254039;
   t1[2310] := -0.1074169;
   t1[2311] := -0.0887473;
   t1[2312] := -0.0695441;
   t1[2313] := -0.0499563;
   t1[2314] := -0.0301329;
   t1[2315] := -0.0102231;
   t1[2316] := 0.0096242;
   t1[2317] := 0.0292598;
   t1[2318] := 0.0485348;
   t1[2319] := 0.0673002;
   t1[2320] := 0.0854068;
   t1[2321] := 0.1027057;
   t1[2322] := 0.1190478;
   t1[2323] := 0.134284;
   t1[2324] := 0.1482654;
   t1[2325] := 0.1608428;
   t1[2326] := 0.1718673;
   t1[2327] := 0.1811903;
   t1[2328] := 0.1887307;
   t1[2329] := 0.1945347;
   t1[2330] := 0.1986626;
   t1[2331] := 0.2011748;
   t1[2332] := 0.2021318;
   t1[2333] := 0.201594;
   t1[2334] := 0.1996216;
   t1[2335] := 0.1962753;
   t1[2336] := 0.1916152;
   t1[2337] := 0.185702;
   t1[2338] := 0.1785959;
   t1[2339] := 0.1703573;
   t1[2340] := 0.1610467;
   t1[2341] := 0.1507245;
   t1[2342] := 0.139451;
   t1[2343] := 0.1272867;
   t1[2344] := 0.1142919;
   t1[2345] := 0.1005271;
   t1[2346] := 0.0860527;
   t1[2347] := 0.0709401;
   t1[2348] := 0.0553158;
   t1[2349] := 0.0393236;
   t1[2350] := -0.4248369;
   t1[2351] := -0.4179277;
   t1[2352] := -0.4100263;
   t1[2353] := -0.401115;
   t1[2354] := -0.3911766;
   t1[2355] := -0.3801935;
   t1[2356] := -0.3681482;
   t1[2357] := -0.3550233;
   t1[2358] := -0.3408041;
   t1[2359] := -0.3255194;
   t1[2360] := -0.3092318;
   t1[2361] := -0.2920052;
   t1[2362] := -0.2739031;
   t1[2363] := -0.2549895;
   t1[2364] := -0.235328;
   t1[2365] := -0.2149823;
   t1[2366] := -0.1940161;
   t1[2367] := -0.1724932;
   t1[2368] := -0.1504773;
   t1[2369] := -0.1280321;
   t1[2370] := -0.1052214;
   t1[2371] := -0.0821088;
   t1[2372] := -0.0587582;
   t1[2373] := -0.0352331;
   t1[2374] := -0.0115973;
   t1[2375] := 0.0120853;
   t1[2376] := 0.0357511;
   t1[2377] := 0.0593363;
   t1[2378] := 0.0827594;
   t1[2379] := 0.105906;
   t1[2380] := 0.1286577;
   t1[2381] := 0.1508963;
   t1[2382] := 0.1725036;
   t1[2383] := 0.1933614;
   t1[2384] := 0.2133514;
   t1[2385] := 0.2323554;
   t1[2386] := 0.2502551;
   t1[2387] := 0.2669323;
   t1[2388] := 0.2822687;
   t1[2389] := 0.2961462;
   t1[2390] := 0.3084463;
   t1[2391] := 0.319051;
   t1[2392] := 0.327842;
   t1[2393] := 0.3347012;
   t1[2394] := 0.3395101;
   t1[2395] := 0.3421504;
   t1[2396] := 0.3425042;
   t1[2397] := 0.3404941;
   t1[2398] := 0.3362485;
   t1[2399] := 0.3299596;
   t1[2400] := 0.3017888;
   t1[2401] := 0.2929916;
   t1[2402] := 0.2837368;
   t1[2403] := 0.2740539;
   t1[2404] := 0.2639727;
   t1[2405] := 0.2535227;
   t1[2406] := 0.2427335;
   t1[2407] := 0.2316348;
   t1[2408] := 0.2202557;
   t1[2409] := 0.2086159;
   t1[2410] := 0.196728;
   t1[2411] := 0.1846043;
   t1[2412] := 0.1722573;
   t1[2413] := 0.1596992;
   t1[2414] := 0.1469425;
   t1[2415] := 0.1339995;
   t1[2416] := 0.1208825;
   t1[2417] := 0.1076039;
   t1[2418] := 0.0941761;
   t1[2419] := 0.0806115;
   t1[2420] := 0.0669224;
   t1[2421] := 0.0531211;
   t1[2422] := 0.03922;
   t1[2423] := 0.0252315;
   t1[2424] := 0.011168;
   t1[2425] := -0.0029583;
   t1[2426] := -0.0171348;
   t1[2427] := -0.0313492;
   t1[2428] := -0.0455605;
   t1[2429] := -0.0596748;
   t1[2430] := -0.0735921;
   t1[2431] := -0.0872125;
   t1[2432] := -0.1004361;
   t1[2433] := -0.1131628;
   t1[2434] := -0.1252928;
   t1[2435] := -0.136726;
   t1[2436] := -0.1473625;
   t1[2437] := -0.1571023;
   t1[2438] := -0.1658456;
   t1[2439] := -0.1734923;
   t1[2440] := -0.1799424;
   t1[2441] := -0.1850961;
   t1[2442] := -0.1888533;
   t1[2443] := -0.1911141;
   t1[2444] := -0.1917786;
   t1[2445] := -0.1907468;
   t1[2446] := -0.1879187;
   t1[2447] := -0.1832308;
   t1[2448] := -0.1768013;
   t1[2449] := -0.1688053;
   t1[2450] := 0.2525824;
   t1[2451] := 0.234157;
   t1[2452] := 0.2152379;
   t1[2453] := 0.1959515;
   t1[2454] := 0.1764241;
   t1[2455] := 0.156782;
   t1[2456] := 0.1371515;
   t1[2457] := 0.1176589;
   t1[2458] := 0.0984263;
   t1[2459] := 0.0795105;
   t1[2460] := 0.0609163;
   t1[2461] := 0.0426475;
   t1[2462] := 0.0247079;
   t1[2463] := 0.007101;
   t1[2464] := -0.0101694;
   t1[2465] := -0.0270996;
   t1[2466] := -0.043686;
   t1[2467] := -0.0599248;
   t1[2468] := -0.0758124;
   t1[2469] := -0.0913451;
   t1[2470] := -0.1065192;
   t1[2471] := -0.121331;
   t1[2472] := -0.1357768;
   t1[2473] := -0.1498529;
   t1[2474] := -0.1635557;
   t1[2475] := -0.1768814;
   t1[2476] := -0.1898264;
   t1[2477] := -0.2023869;
   t1[2478] := -0.2145509;
   t1[2479] := -0.2262909;
   t1[2480] := -0.2375775;
   t1[2481] := -0.2483814;
   t1[2482] := -0.2586735;
   t1[2483] := -0.2684242;
   t1[2484] := -0.2776044;
   t1[2485] := -0.2861848;
   t1[2486] := -0.2941359;
   t1[2487] := -0.3014286;
   t1[2488] := -0.3080335;
   t1[2489] := -0.3139214;
   t1[2490] := -0.3190629;
   t1[2491] := -0.3234286;
   t1[2492] := -0.3269894;
   t1[2493] := -0.3297159;
   t1[2494] := -0.3315789;
   t1[2495] := -0.3325488;
   t1[2496] := -0.3325966;
   t1[2497] := -0.3317031;
   t1[2498] := -0.3298996;
   t1[2499] := -0.3272333;
   t1[2500] := 0.1863346;
   t1[2501] := 0.1800162;
   t1[2502] := 0.1729414;
   t1[2503] := 0.1650857;
   t1[2504] := 0.1564246;
   t1[2505] := 0.1469336;
   t1[2506] := 0.1365881;
   t1[2507] := 0.1253638;
   t1[2508] := 0.1132393;
   t1[2509] := 0.1002423;
   t1[2510] := 0.0864392;
   t1[2511] := 0.0718976;
   t1[2512] := 0.0566846;
   t1[2513] := 0.0408679;
   t1[2514] := 0.0245148;
   t1[2515] := 0.0076928;
   t1[2516] := -0.0095309;
   t1[2517] := -0.0270886;
   t1[2518] := -0.044913;
   t1[2519] := -0.0629367;
   t1[2520] := -0.0810922;
   t1[2521] := -0.0993121;
   t1[2522] := -0.1175291;
   t1[2523] := -0.1356757;
   t1[2524] := -0.1536844;
   t1[2525] := -0.1714878;
   t1[2526] := -0.1890186;
   t1[2527] := -0.2062093;
   t1[2528] := -0.2229935;
   t1[2529] := -0.2393069;
   t1[2530] := -0.2550855;
   t1[2531] := -0.2702649;
   t1[2532] := -0.2847811;
   t1[2533] := -0.2985701;
   t1[2534] := -0.3115676;
   t1[2535] := -0.3237095;
   t1[2536] := -0.3349317;
   t1[2537] := -0.3451701;
   t1[2538] := -0.3543605;
   t1[2539] := -0.3624389;
   t1[2540] := -0.369341;
   t1[2541] := -0.3750027;
   t1[2542] := -0.37936;
   t1[2543] := -0.3823487;
   t1[2544] := -0.3839047;
   t1[2545] := -0.3839638;
   t1[2546] := -0.3824619;
   t1[2547] := -0.3793586;
   t1[2548] := -0.3747315;
   t1[2549] := -0.3686952;
   t1[2550] := 0.0815692;
   t1[2551] := 0.0721724;
   t1[2552] := 0.0627858;
   t1[2553] := 0.0534844;
   t1[2554] := 0.0443431;
   t1[2555] := 0.0354371;
   t1[2556] := 0.0268412;
   t1[2557] := 0.0186305;
   t1[2558] := 0.0108776;
   t1[2559] := 0.0036155;
   t1[2560] := -0.0031535;
   t1[2561] := -0.0094281;
   t1[2562] := -0.0152069;
   t1[2563] := -0.0204886;
   t1[2564] := -0.0252718;
   t1[2565] := -0.029555;
   t1[2566] := -0.0333371;
   t1[2567] := -0.0366166;
   t1[2568] := -0.0393921;
   t1[2569] := -0.0416622;
   t1[2570] := -0.0434257;
   t1[2571] := -0.0446811;
   t1[2572] := -0.0454271;
   t1[2573] := -0.0456624;
   t1[2574] := -0.0453855;
   t1[2575] := -0.044595;
   t1[2576] := -0.0432897;
   t1[2577] := -0.0414683;
   t1[2578] := -0.039138;
   t1[2579] := -0.0363222;
   t1[2580] := -0.0330463;
   t1[2581] := -0.0293356;
   t1[2582] := -0.0252153;
   t1[2583] := -0.0207107;
   t1[2584] := -0.0158472;
   t1[2585] := -0.0106499;
   t1[2586] := -0.0051443;
   t1[2587] := 0.0006445;
   t1[2588] := 0.0066911;
   t1[2589] := 0.0129702;
   t1[2590] := 0.0194567;
   t1[2591] := 0.026125;
   t1[2592] := 0.0329501;
   t1[2593] := 0.0399066;
   t1[2594] := 0.0469692;
   t1[2595] := 0.0541127;
   t1[2596] := 0.0613117;
   t1[2597] := 0.0685377;
   t1[2598] := 0.0757459;
   t1[2599] := 0.0828866;
   t1[2600] := 0.0296985;
   t1[2601] := 0.0298958;
   t1[2602] := 0.0298572;
   t1[2603] := 0.0295598;
   t1[2604] := 0.0289804;
   t1[2605] := 0.028096;
   t1[2606] := 0.0268834;
   t1[2607] := 0.0253197;
   t1[2608] := 0.0233825;
   t1[2609] := 0.0210612;
   t1[2610] := 0.0183545;
   t1[2611] := 0.0152612;
   t1[2612] := 0.0117802;
   t1[2613] := 0.0079105;
   t1[2614] := 0.0036509;
   t1[2615] := -0.0009996;
   t1[2616] := -0.0060423;
   t1[2617] := -0.0114781;
   t1[2618] := -0.0173083;
   t1[2619] := -0.0235339;
   t1[2620] := -0.030156;
   t1[2621] := -0.0371757;
   t1[2622] := -0.0445942;
   t1[2623] := -0.0524126;
   t1[2624] := -0.0606318;
   t1[2625] := -0.0692532;
   t1[2626] := -0.0782777;
   t1[2627] := -0.0877063;
   t1[2628] := -0.0975138;
   t1[2629] := -0.1076262;
   t1[2630] := -0.1179638;
   t1[2631] := -0.1284467;
   t1[2632] := -0.1389955;
   t1[2633] := -0.1495303;
   t1[2634] := -0.1599716;
   t1[2635] := -0.1702395;
   t1[2636] := -0.1802546;
   t1[2637] := -0.189937;
   t1[2638] := -0.1992071;
   t1[2639] := -0.2079852;
   t1[2640] := -0.2161917;
   t1[2641] := -0.2237468;
   t1[2642] := -0.230571;
   t1[2643] := -0.2365844;
   t1[2644] := -0.2417075;
   t1[2645] := -0.2458604;
   t1[2646] := -0.2489637;
   t1[2647] := -0.2509559;
   t1[2648] := -0.2518681;
   t1[2649] := -0.2517596;
   t1[2650] := 0.2789594;
   t1[2651] := 0.2709424;
   t1[2652] := 0.2617649;
   t1[2653] := 0.2513233;
   t1[2654] := 0.2395139;
   t1[2655] := 0.2262332;
   t1[2656] := 0.2113774;
   t1[2657] := 0.1948428;
   t1[2658] := 0.1765366;
   t1[2659] := 0.1565279;
   t1[2660] := 0.135014;
   t1[2661] := 0.1121957;
   t1[2662] := 0.0882736;
   t1[2663] := 0.0634485;
   t1[2664] := 0.0379211;
   t1[2665] := 0.0118922;
   t1[2666] := -0.0144376;
   t1[2667] := -0.0408675;
   t1[2668] := -0.0671968;
   t1[2669] := -0.0932248;
   t1[2670] := -0.1187508;
   t1[2671] := -0.1435741;
   t1[2672] := -0.1674938;
   t1[2673] := -0.1903095;
   t1[2674] := -0.2118202;
   t1[2675] := -0.2318252;
   t1[2676] := -0.2501238;
   t1[2677] := -0.2665164;
   t1[2678] := -0.2809054;
   t1[2679] := -0.2933874;
   t1[2680] := -0.304081;
   t1[2681] := -0.3131043;
   t1[2682] := -0.3205758;
   t1[2683] := -0.3266138;
   t1[2684] := -0.3313366;
   t1[2685] := -0.3348626;
   t1[2686] := -0.3373102;
   t1[2687] := -0.3387977;
   t1[2688] := -0.3394434;
   t1[2689] := -0.3393657;
   t1[2690] := -0.3386829;
   t1[2691] := -0.3375134;
   t1[2692] := -0.3359756;
   t1[2693] := -0.3341878;
   t1[2694] := -0.3322684;
   t1[2695] := -0.3303355;
   t1[2696] := -0.3285078;
   t1[2697] := -0.32688;
   t1[2698] := -0.3254305;
   t1[2699] := -0.3241007;
   t1[2700] := -0.0089786;
   t1[2701] := -0.0170903;
   t1[2702] := -0.0249782;
   t1[2703] := -0.0325892;
   t1[2704] := -0.0398705;
   t1[2705] := -0.046769;
   t1[2706] := -0.0532318;
   t1[2707] := -0.0592059;
   t1[2708] := -0.0646412;
   t1[2709] := -0.069531;
   t1[2710] := -0.0739032;
   t1[2711] := -0.0777865;
   t1[2712] := -0.0812096;
   t1[2713] := -0.0842011;
   t1[2714] := -0.0867897;
   t1[2715] := -0.0890041;
   t1[2716] := -0.090873;
   t1[2717] := -0.0924251;
   t1[2718] := -0.0936891;
   t1[2719] := -0.0946936;
   t1[2720] := -0.0954674;
   t1[2721] := -0.0960391;
   t1[2722] := -0.0964375;
   t1[2723] := -0.0966911;
   t1[2724] := -0.0968288;
   t1[2725] := -0.0968791;
   t1[2726] := -0.0968709;
   t1[2727] := -0.0968326;
   t1[2728] := -0.0967854;
   t1[2729] := -0.0967358;
   t1[2730] := -0.096689;
   t1[2731] := -0.09665;
   t1[2732] := -0.0966238;
   t1[2733] := -0.0966156;
   t1[2734] := -0.0966302;
   t1[2735] := -0.0966729;
   t1[2736] := -0.0967486;
   t1[2737] := -0.0968624;
   t1[2738] := -0.0970193;
   t1[2739] := -0.0972244;
   t1[2740] := -0.0974828;
   t1[2741] := -0.0977994;
   t1[2742] := -0.0981794;
   t1[2743] := -0.0986278;
   t1[2744] := -0.0991497;
   t1[2745] := -0.09975;
   t1[2746] := -0.1004339;
   t1[2747] := -0.1012022;
   t1[2748] := -0.1020352;
   t1[2749] := -0.1029065;
   t1[2750] := 0.1839082;
   t1[2751] := 0.1719079;
   t1[2752] := 0.1598567;
   t1[2753] := 0.1477929;
   t1[2754] := 0.1357548;
   t1[2755] := 0.1237808;
   t1[2756] := 0.111909;
   t1[2757] := 0.1001777;
   t1[2758] := 0.0886241;
   t1[2759] := 0.077267;
   t1[2760] := 0.0661109;
   t1[2761] := 0.0551598;
   t1[2762] := 0.0444179;
   t1[2763] := 0.0338891;
   t1[2764] := 0.0235777;
   t1[2765] := 0.0134876;
   t1[2766] := 0.0036229;
   t1[2767] := -0.0060122;
   t1[2768] := -0.0154137;
   t1[2769] := -0.0245775;
   t1[2770] := -0.0334996;
   t1[2771] := -0.0421758;
   t1[2772] := -0.0506021;
   t1[2773] := -0.0587744;
   t1[2774] := -0.0666886;
   t1[2775] := -0.0743406;
   t1[2776] := -0.0817264;
   t1[2777] := -0.088842;
   t1[2778] := -0.0956898;
   t1[2779] := -0.1022846;
   t1[2780] := -0.1086426;
   t1[2781] := -0.1147801;
   t1[2782] := -0.1207133;
   t1[2783] := -0.1264583;
   t1[2784] := -0.1320314;
   t1[2785] := -0.1374487;
   t1[2786] := -0.1427265;
   t1[2787] := -0.1478809;
   t1[2788] := -0.1529282;
   t1[2789] := -0.1578846;
   t1[2790] := -0.1627663;
   t1[2791] := -0.1675894;
   t1[2792] := -0.1723702;
   t1[2793] := -0.1771248;
   t1[2794] := -0.1818696;
   t1[2795] := -0.1866206;
   t1[2796] := -0.1913941;
   t1[2797] := -0.1961968;
   t1[2798] := -0.2009879;
   t1[2799] := -0.2057118;
   t1[2800] := 0.129127;
   t1[2801] := 0.1244142;
   t1[2802] := 0.1193461;
   t1[2803] := 0.1139074;
   t1[2804] := 0.1080832;
   t1[2805] := 0.1018582;
   t1[2806] := 0.0952174;
   t1[2807] := 0.0881457;
   t1[2808] := 0.0806309;
   t1[2809] := 0.0727068;
   t1[2810] := 0.0644431;
   t1[2811] := 0.0559105;
   t1[2812] := 0.0471798;
   t1[2813] := 0.0383219;
   t1[2814] := 0.0294074;
   t1[2815] := 0.0205071;
   t1[2816] := 0.0116917;
   t1[2817] := 0.0030321;
   t1[2818] := -0.0054011;
   t1[2819] := -0.0135371;
   t1[2820] := -0.021305;
   t1[2821] := -0.0286343;
   t1[2822] := -0.035454;
   t1[2823] := -0.0416934;
   t1[2824] := -0.0472819;
   t1[2825] := -0.0521486;
   t1[2826] := -0.0562227;
   t1[2827] := -0.059434;
   t1[2828] := -0.0617627;
   t1[2829] := -0.0632845;
   t1[2830] := -0.0640861;
   t1[2831] := -0.0642538;
   t1[2832] := -0.0638743;
   t1[2833] := -0.0630341;
   t1[2834] := -0.0618197;
   t1[2835] := -0.0603176;
   t1[2836] := -0.0586143;
   t1[2837] := -0.0567965;
   t1[2838] := -0.0549505;
   t1[2839] := -0.053163;
   t1[2840] := -0.0515205;
   t1[2841] := -0.0501094;
   t1[2842] := -0.0490163;
   t1[2843] := -0.0483278;
   t1[2844] := -0.0481303;
   t1[2845] := -0.0485104;
   t1[2846] := -0.0495547;
   t1[2847] := -0.051326;
   t1[2848] := -0.0537697;
   t1[2849] := -0.0567943;
   t1[2850] := 0.1542486;
   t1[2851] := 0.1550493;
   t1[2852] := 0.1557622;
   t1[2853] := 0.1563427;
   t1[2854] := 0.1567464;
   t1[2855] := 0.1569286;
   t1[2856] := 0.1568447;
   t1[2857] := 0.1564502;
   t1[2858] := 0.1557015;
   t1[2859] := 0.15457;
   t1[2860] := 0.1530392;
   t1[2861] := 0.1510926;
   t1[2862] := 0.1487141;
   t1[2863] := 0.1458872;
   t1[2864] := 0.1425956;
   t1[2865] := 0.138823;
   t1[2866] := 0.1345531;
   t1[2867] := 0.1297696;
   t1[2868] := 0.1244561;
   t1[2869] := 0.1185963;
   t1[2870] := 0.1121739;
   t1[2871] := 0.1051726;
   t1[2872] := 0.097576;
   t1[2873] := 0.0893678;
   t1[2874] := 0.0805317;
   t1[2875] := 0.0710514;
   t1[2876] := 0.0609105;
   t1[2877] := 0.0500932;
   t1[2878] := 0.0386272;
   t1[2879] := 0.0266233;
   t1[2880] := 0.0142016;
   t1[2881] := 0.0014821;
   t1[2882] := -0.0114151;
   t1[2883] := -0.02437;
   t1[2884] := -0.0372626;
   t1[2885] := -0.0499728;
   t1[2886] := -0.0623805;
   t1[2887] := -0.0743657;
   t1[2888] := -0.0858084;
   t1[2889] := -0.0965885;
   t1[2890] := -0.106586;
   t1[2891] := -0.1156808;
   t1[2892] := -0.1237528;
   t1[2893] := -0.1306822;
   t1[2894] := -0.1363487;
   t1[2895] := -0.1406323;
   t1[2896] := -0.143413;
   t1[2897] := -0.1445999;
   t1[2898] := -0.1442478;
   t1[2899] := -0.1424568;
   t1[2900] := 0.2432433;
   t1[2901] := 0.2353556;
   t1[2902] := 0.2270421;
   t1[2903] := 0.2183365;
   t1[2904] := 0.209273;
   t1[2905] := 0.1998853;
   t1[2906] := 0.1902075;
   t1[2907] := 0.1802735;
   t1[2908] := 0.1701179;
   t1[2909] := 0.1597853;
   t1[2910] := 0.1493282;
   t1[2911] := 0.1387992;
   t1[2912] := 0.128251;
   t1[2913] := 0.1177363;
   t1[2914] := 0.1073077;
   t1[2915] := 0.097018;
   t1[2916] := 0.0869198;
   t1[2917] := 0.0770657;
   t1[2918] := 0.0675085;
   t1[2919] := 0.0583008;
   t1[2920] := 0.0494953;
   t1[2921] := 0.0411446;
   t1[2922] := 0.0333014;
   t1[2923] := 0.0260185;
   t1[2924] := 0.0193484;
   t1[2925] := 0.0133438;
   t1[2926] := 0.0080575;
   t1[2927] := 0.0035418;
   t1[2928] := -0.0001807;
   t1[2929] := -0.0031441;
   t1[2930] := -0.0053886;
   t1[2931] := -0.0069547;
   t1[2932] := -0.0078826;
   t1[2933] := -0.0082128;
   t1[2934] := -0.0079854;
   t1[2935] := -0.007241;
   t1[2936] := -0.0060198;
   t1[2937] := -0.0043621;
   t1[2938] := -0.0023084;
   t1[2939] := 0.0001011;
   t1[2940] := 0.0028261;
   t1[2941] := 0.0058261;
   t1[2942] := 0.0090608;
   t1[2943] := 0.01249;
   t1[2944] := 0.0160732;
   t1[2945] := 0.0197702;
   t1[2946] := 0.0235405;
   t1[2947] := 0.027347;
   t1[2948] := 0.0311682;
   t1[2949] := 0.0349876;
   t1[2950] := 0.0060134;
   t1[2951] := 0.0075953;
   t1[2952] := 0.0095188;
   t1[2953] := 0.01177;
   t1[2954] := 0.0143348;
   t1[2955] := 0.017199;
   t1[2956] := 0.0203486;
   t1[2957] := 0.0237696;
   t1[2958] := 0.0274472;
   t1[2959] := 0.0313589;
   t1[2960] := 0.0354757;
   t1[2961] := 0.0397684;
   t1[2962] := 0.0442078;
   t1[2963] := 0.0487648;
   t1[2964] := 0.0534102;
   t1[2965] := 0.0581149;
   t1[2966] := 0.0628497;
   t1[2967] := 0.0675854;
   t1[2968] := 0.0722929;
   t1[2969] := 0.076943;
   t1[2970] := 0.0815065;
   t1[2971] := 0.0859543;
   t1[2972] := 0.0902573;
   t1[2973] := 0.0943862;
   t1[2974] := 0.0983119;
   t1[2975] := 0.1020052;
   t1[2976] := 0.105437;
   t1[2977] := 0.1085783;
   t1[2978] := 0.111415;
   t1[2979] := 0.1139619;
   t1[2980] := 0.1162366;
   t1[2981] := 0.118257;
   t1[2982] := 0.1200409;
   t1[2983] := 0.121606;
   t1[2984] := 0.1229703;
   t1[2985] := 0.1241514;
   t1[2986] := 0.1251671;
   t1[2987] := 0.1260353;
   t1[2988] := 0.1267737;
   t1[2989] := 0.1274002;
   t1[2990] := 0.1279325;
   t1[2991] := 0.1283884;
   t1[2992] := 0.1287857;
   t1[2993] := 0.1291423;
   t1[2994] := 0.1294759;
   t1[2995] := 0.1298042;
   t1[2996] := 0.1301452;
   t1[2997] := 0.1305105;
   t1[2998] := 0.1308815;
   t1[2999] := 0.1312302;
   t1[3000] := 0.1256087;
   t1[3001] := 0.1352973;
   t1[3002] := 0.1443325;
   t1[3003] := 0.152559;
   t1[3004] := 0.1598216;
   t1[3005] := 0.165965;
   t1[3006] := 0.170834;
   t1[3007] := 0.1742733;
   t1[3008] := 0.1761368;
   t1[3009] := 0.1764177;
   t1[3010] := 0.1752191;
   t1[3011] := 0.1726473;
   t1[3012] := 0.1688082;
   t1[3013] := 0.163808;
   t1[3014] := 0.1577529;
   t1[3015] := 0.1507489;
   t1[3016] := 0.1429021;
   t1[3017] := 0.1343186;
   t1[3018] := 0.1251047;
   t1[3019] := 0.1153662;
   t1[3020] := 0.1052095;
   t1[3021] := 0.0947405;
   t1[3022] := 0.0840654;
   t1[3023] := 0.0732903;
   t1[3024] := 0.0625214;
   t1[3025] := 0.0518646;
   t1[3026] := 0.0414262;
   t1[3027] := 0.0313121;
   t1[3028] := 0.0216062;
   t1[3029] := 0.0123507;
   t1[3030] := 0.0035835;
   t1[3031] := -0.0046578;
   t1[3032] := -0.0123355;
   t1[3033] := -0.019412;
   t1[3034] := -0.0258496;
   t1[3035] := -0.0316105;
   t1[3036] := -0.0366572;
   t1[3037] := -0.0409519;
   t1[3038] := -0.0444569;
   t1[3039] := -0.0471346;
   t1[3040] := -0.0489473;
   t1[3041] := -0.0498573;
   t1[3042] := -0.049827;
   t1[3043] := -0.0488186;
   t1[3044] := -0.0467944;
   t1[3045] := -0.0437169;
   t1[3046] := -0.0395483;
   t1[3047] := -0.0342693;
   t1[3048] := -0.0279528;
   t1[3049] := -0.0207005;
   t1[3050] := 0.0231812;
   t1[3051] := 0.0164768;
   t1[3052] := 0.0097991;
   t1[3053] := 0.0031845;
   t1[3054] := -0.0033309;
   t1[3055] := -0.009711;
   t1[3056] := -0.0159195;
   t1[3057] := -0.0219202;
   t1[3058] := -0.0276777;
   t1[3059] := -0.0331666;
   t1[3060] := -0.0383697;
   t1[3061] := -0.0432701;
   t1[3062] := -0.0478508;
   t1[3063] := -0.0520948;
   t1[3064] := -0.0559851;
   t1[3065] := -0.0595047;
   t1[3066] := -0.0626367;
   t1[3067] := -0.0653641;
   t1[3068] := -0.0676698;
   t1[3069] := -0.0695369;
   t1[3070] := -0.0709485;
   t1[3071] := -0.0718874;
   t1[3072] := -0.0723369;
   t1[3073] := -0.0722798;
   t1[3074] := -0.0716991;
   t1[3075] := -0.070578;
   t1[3076] := -0.0688994;
   t1[3077] := -0.0666465;
   t1[3078] := -0.0638269;
   t1[3079] := -0.0604939;
   t1[3080] := -0.0567063;
   t1[3081] := -0.0525226;
   t1[3082] := -0.0480013;
   t1[3083] := -0.0432012;
   t1[3084] := -0.0381807;
   t1[3085] := -0.0329986;
   t1[3086] := -0.0277133;
   t1[3087] := -0.0223835;
   t1[3088] := -0.0170678;
   t1[3089] := -0.0118248;
   t1[3090] := -0.0067131;
   t1[3091] := -0.0017912;
   t1[3092] := 0.0028822;
   t1[3093] := 0.0072485;
   t1[3094] := 0.0112491;
   t1[3095] := 0.0148255;
   t1[3096] := 0.017919;
   t1[3097] := 0.020481;
   t1[3098] := 0.022513;
   t1[3099] := 0.0240322;
   t1[3100] := -0.038803;
   t1[3101] := -0.041465;
   t1[3102] := -0.0442218;
   t1[3103] := -0.0471058;
   t1[3104] := -0.050149;
   t1[3105] := -0.0533837;
   t1[3106] := -0.0568421;
   t1[3107] := -0.0605563;
   t1[3108] := -0.0645558;
   t1[3109] := -0.0688262;
   t1[3110] := -0.0733187;
   t1[3111] := -0.0779837;
   t1[3112] := -0.0827715;
   t1[3113] := -0.0876325;
   t1[3114] := -0.0925168;
   t1[3115] := -0.097375;
   t1[3116] := -0.1021573;
   t1[3117] := -0.106814;
   t1[3118] := -0.1112955;
   t1[3119] := -0.115552;
   t1[3120] := -0.119534;
   t1[3121] := -0.1231917;
   t1[3122] := -0.1264755;
   t1[3123] := -0.1293356;
   t1[3124] := -0.1317225;
   t1[3125] := -0.1335863;
   t1[3126] := -0.1348776;
   t1[3127] := -0.1355469;
   t1[3128] := -0.1355845;
   t1[3129] := -0.135056;
   t1[3130] := -0.1340351;
   t1[3131] := -0.1325956;
   t1[3132] := -0.1308115;
   t1[3133] := -0.1287565;
   t1[3134] := -0.1265045;
   t1[3135] := -0.1241293;
   t1[3136] := -0.1217048;
   t1[3137] := -0.1193047;
   t1[3138] := -0.117003;
   t1[3139] := -0.1148734;
   t1[3140] := -0.1129898;
   t1[3141] := -0.111426;
   t1[3142] := -0.1102559;
   t1[3143] := -0.1095533;
   t1[3144] := -0.109392;
   t1[3145] := -0.1098459;
   t1[3146] := -0.1109888;
   t1[3147] := -0.112873;
   t1[3148] := -0.1154429;
   t1[3149] := -0.1186093;
   t1[3150] := 0.0876806;
   t1[3151] := 0.0804098;
   t1[3152] := 0.0733107;
   t1[3153] := 0.0664517;
   t1[3154] := 0.0599012;
   t1[3155] := 0.0537276;
   t1[3156] := 0.0479992;
   t1[3157] := 0.0427845;
   t1[3158] := 0.0381484;
   t1[3159] := 0.0341009;
   t1[3160] := 0.0306092;
   t1[3161] := 0.027639;
   t1[3162] := 0.0251565;
   t1[3163] := 0.0231273;
   t1[3164] := 0.0215176;
   t1[3165] := 0.020293;
   t1[3166] := 0.0194197;
   t1[3167] := 0.0188633;
   t1[3168] := 0.01859;
   t1[3169] := 0.0185655;
   t1[3170] := 0.0187558;
   t1[3171] := 0.0191267;
   t1[3172] := 0.0196442;
   t1[3173] := 0.0202742;
   t1[3174] := 0.0209826;
   t1[3175] := 0.0217353;
   t1[3176] := 0.0224981;
   t1[3177] := 0.0232371;
   t1[3178] := 0.0239225;
   t1[3179] := 0.0245327;
   t1[3180] := 0.0250472;
   t1[3181] := 0.0254454;
   t1[3182] := 0.0257066;
   t1[3183] := 0.0258103;
   t1[3184] := 0.0257358;
   t1[3185] := 0.0254626;
   t1[3186] := 0.0249699;
   t1[3187] := 0.0242373;
   t1[3188] := 0.0232441;
   t1[3189] := 0.0219697;
   t1[3190] := 0.0203935;
   t1[3191] := 0.0184949;
   t1[3192] := 0.0162533;
   t1[3193] := 0.013648;
   t1[3194] := 0.0106585;
   t1[3195] := 0.0072642;
   t1[3196] := 0.0034444;
   t1[3197] := -0.0008121;
   t1[3198] := -0.0054704;
   t1[3199] := -0.0104808;
   t1[3200] := 0.156688;
   t1[3201] := 0.1584898;
   t1[3202] := 0.1597388;
   t1[3203] := 0.1603476;
   t1[3204] := 0.1602288;
   t1[3205] := 0.159295;
   t1[3206] := 0.1574585;
   t1[3207] := 0.154632;
   t1[3208] := 0.1507343;
   t1[3209] := 0.1457798;
   t1[3210] := 0.1398588;
   t1[3211] := 0.1330631;
   t1[3212] := 0.1254851;
   t1[3213] := 0.1172166;
   t1[3214] := 0.1083499;
   t1[3215] := 0.098977;
   t1[3216] := 0.08919;
   t1[3217] := 0.0790811;
   t1[3218] := 0.0687422;
   t1[3219] := 0.0582655;
   t1[3220] := 0.047743;
   t1[3221] := 0.037267;
   t1[3222] := 0.0269294;
   t1[3223] := 0.0168223;
   t1[3224] := 0.0070378;
   t1[3225] := -0.0023319;
   t1[3226] := -0.0111948;
   t1[3227] := -0.0194591;
   t1[3228] := -0.0270664;
   t1[3229] := -0.0340217;
   t1[3230] := -0.0403372;
   t1[3231] := -0.0460248;
   t1[3232] := -0.0510966;
   t1[3233] := -0.0555648;
   t1[3234] := -0.0594414;
   t1[3235] := -0.0627384;
   t1[3236] := -0.0654681;
   t1[3237] := -0.0676423;
   t1[3238] := -0.0692732;
   t1[3239] := -0.0703729;
   t1[3240] := -0.0709534;
   t1[3241] := -0.0710269;
   t1[3242] := -0.0706053;
   t1[3243] := -0.0697009;
   t1[3244] := -0.0683255;
   t1[3245] := -0.0664914;
   t1[3246] := -0.0642106;
   t1[3247] := -0.0614983;
   t1[3248] := -0.0583853;
   t1[3249] := -0.0549072;
   t1[3250] := -0.031862;
   t1[3251] := -0.035804;
   t1[3252] := -0.039725;
   t1[3253] := -0.0436243;
   t1[3254] := -0.0475011;
   t1[3255] := -0.0513548;
   t1[3256] := -0.0551847;
   t1[3257] := -0.05899;
   t1[3258] := -0.0627687;
   t1[3259] := -0.0664977;
   t1[3260] := -0.0701374;
   t1[3261] := -0.0736476;
   t1[3262] := -0.0769884;
   t1[3263] := -0.0801197;
   t1[3264] := -0.0830013;
   t1[3265] := -0.0855932;
   t1[3266] := -0.0878554;
   t1[3267] := -0.0897477;
   t1[3268] := -0.0912301;
   t1[3269] := -0.0922625;
   t1[3270] := -0.0928049;
   t1[3271] := -0.0928171;
   t1[3272] := -0.0922591;
   t1[3273] := -0.0910909;
   t1[3274] := -0.0892723;
   t1[3275] := -0.0867632;
   t1[3276] := -0.0835237;
   t1[3277] := -0.0795138;
   t1[3278] := -0.0747269;
   t1[3279] := -0.0692185;
   t1[3280] := -0.063051;
   t1[3281] := -0.0562872;
   t1[3282] := -0.0489895;
   t1[3283] := -0.0412205;
   t1[3284] := -0.0330428;
   t1[3285] := -0.024519;
   t1[3286] := -0.0157115;
   t1[3287] := -0.0066831;
   t1[3288] := 0.0025039;
   t1[3289] := 0.0117868;
   t1[3290] := 0.021103;
   t1[3291] := 0.0303901;
   t1[3292] := 0.0395853;
   t1[3293] := 0.0486263;
   t1[3294] := 0.0574503;
   t1[3295] := 0.0659949;
   t1[3296] := 0.0741974;
   t1[3297] := 0.0820048;
   t1[3298] := 0.0894105;
   t1[3299] := 0.0964227;
   t1[3300] := -0.0839461;
   t1[3301] := -0.0761973;
   t1[3302] := -0.0686025;
   t1[3303] := -0.0612328;
   t1[3304] := -0.0541593;
   t1[3305] := -0.047453;
   t1[3306] := -0.041185;
   t1[3307] := -0.0354264;
   t1[3308] := -0.0302436;
   t1[3309] := -0.0256303;
   t1[3310] := -0.0215232;
   t1[3311] := -0.0178572;
   t1[3312] := -0.0145674;
   t1[3313] := -0.0115889;
   t1[3314] := -0.0088567;
   t1[3315] := -0.0063059;
   t1[3316] := -0.0038716;
   t1[3317] := -0.0014887;
   t1[3318] := 0.0009077;
   t1[3319] := 0.0033825;
   t1[3320] := 0.0060006;
   t1[3321] := 0.0088271;
   t1[3322] := 0.0119268;
   t1[3323] := 0.0153648;
   t1[3324] := 0.0192059;
   t1[3325] := 0.0235151;
   t1[3326] := 0.0283574;
   t1[3327] := 0.0337973;
   t1[3328] := 0.0398612;
   t1[3329] := 0.0465024;
   t1[3330] := 0.0536664;
   t1[3331] := 0.0612984;
   t1[3332] := 0.069344;
   t1[3333] := 0.0777483;
   t1[3334] := 0.0864569;
   t1[3335] := 0.0954149;
   t1[3336] := 0.1045679;
   t1[3337] := 0.1138611;
   t1[3338] := 0.1232399;
   t1[3339] := 0.1326497;
   t1[3340] := 0.1420359;
   t1[3341] := 0.1513437;
   t1[3342] := 0.1605185;
   t1[3343] := 0.1695058;
   t1[3344] := 0.1782509;
   t1[3345] := 0.1866991;
   t1[3346] := 0.1947958;
   t1[3347] := 0.2024895;
   t1[3348] := 0.2097449;
   t1[3349] := 0.2165315;
   t1[3350] := -0.0905587;
   t1[3351] := -0.0872743;
   t1[3352] := -0.0835619;
   t1[3353] := -0.0793684;
   t1[3354] := -0.0746408;
   t1[3355] := -0.0693258;
   t1[3356] := -0.0633704;
   t1[3357] := -0.0567213;
   t1[3358] := -0.0493303;
   t1[3359] := -0.041221;
   t1[3360] := -0.0324741;
   t1[3361] := -0.0231717;
   t1[3362] := -0.0133961;
   t1[3363] := -0.0032293;
   t1[3364] := 0.0072464;
   t1[3365] := 0.0179488;
   t1[3366] := 0.0287959;
   t1[3367] := 0.0397053;
   t1[3368] := 0.0505951;
   t1[3369] := 0.0613829;
   t1[3370] := 0.0719866;
   t1[3371] := 0.0823241;
   t1[3372] := 0.0923131;
   t1[3373] := 0.1018716;
   t1[3374] := 0.1109173;
   t1[3375] := 0.119368;
   t1[3376] := 0.1271416;
   t1[3377] := 0.1341563;
   t1[3378] := 0.1403646;
   t1[3379] := 0.1457842;
   t1[3380] := 0.1504402;
   t1[3381] := 0.1543578;
   t1[3382] := 0.157562;
   t1[3383] := 0.1600779;
   t1[3384] := 0.1619305;
   t1[3385] := 0.163145;
   t1[3386] := 0.1637464;
   t1[3387] := 0.1637598;
   t1[3388] := 0.1632102;
   t1[3389] := 0.1621228;
   t1[3390] := 0.1605227;
   t1[3391] := 0.1584348;
   t1[3392] := 0.1558844;
   t1[3393] := 0.1528964;
   t1[3394] := 0.1494959;
   t1[3395] := 0.1457081;
   t1[3396] := 0.141558;
   t1[3397] := 0.1370706;
   t1[3398] := 0.1322715;
   t1[3399] := 0.127186;
   t1[3400] := 0.0801389;
   t1[3401] := 0.0851319;
   t1[3402] := 0.0898563;
   t1[3403] := 0.0942865;
   t1[3404] := 0.0983973;
   t1[3405] := 0.1021633;
   t1[3406] := 0.105559;
   t1[3407] := 0.108559;
   t1[3408] := 0.1111395;
   t1[3409] := 0.1132981;
   t1[3410] := 0.1150501;
   t1[3411] := 0.1164108;
   t1[3412] := 0.1173959;
   t1[3413] := 0.1180208;
   t1[3414] := 0.118301;
   t1[3415] := 0.1182521;
   t1[3416] := 0.1178895;
   t1[3417] := 0.1172288;
   t1[3418] := 0.1162854;
   t1[3419] := 0.115075;
   t1[3420] := 0.113613;
   t1[3421] := 0.1119149;
   t1[3422] := 0.1099962;
   t1[3423] := 0.1078724;
   t1[3424] := 0.1055591;
   t1[3425] := 0.1030718;
   t1[3426] := 0.100426;
   t1[3427] := 0.097637;
   t1[3428] := 0.0947118;
   t1[3429] := 0.0916409;
   t1[3430] := 0.0884129;
   t1[3431] := 0.0850164;
   t1[3432] := 0.0814403;
   t1[3433] := 0.0776731;
   t1[3434] := 0.0737036;
   t1[3435] := 0.0695204;
   t1[3436] := 0.0651121;
   t1[3437] := 0.0604676;
   t1[3438] := 0.0555754;
   t1[3439] := 0.0504243;
   t1[3440] := 0.0450029;
   t1[3441] := 0.0392999;
   t1[3442] := 0.033304;
   t1[3443] := 0.0270039;
   t1[3444] := 0.0203882;
   t1[3445] := 0.0134456;
   t1[3446] := 0.0061649;
   t1[3447] := -0.0014545;
   t1[3448] := -0.0093581;
   t1[3449] := -0.0174747;
   t1[3450] := -0.1516485;
   t1[3451] := -0.1532073;
   t1[3452] := -0.154109;
   t1[3453] := -0.1542937;
   t1[3454] := -0.1537017;
   t1[3455] := -0.1522733;
   t1[3456] := -0.1499484;
   t1[3457] := -0.1466674;
   t1[3458] := -0.1423761;
   t1[3459] := -0.1371075;
   t1[3460] := -0.1309636;
   t1[3461] := -0.124048;
   t1[3462] := -0.1164644;
   t1[3463] := -0.1083164;
   t1[3464] := -0.0997078;
   t1[3465] := -0.0907423;
   t1[3466] := -0.0815235;
   t1[3467] := -0.0721551;
   t1[3468] := -0.0627407;
   t1[3469] := -0.0533842;
   t1[3470] := -0.0441891;
   t1[3471] := -0.0352591;
   t1[3472] := -0.026698;
   t1[3473] := -0.0186094;
   t1[3474] := -0.0110969;
   t1[3475] := -0.0042644;
   t1[3476] := 0.0017847;
   t1[3477] := 0.0069469;
   t1[3478] := 0.0111756;
   t1[3479] := 0.0145306;
   t1[3480] := 0.0170836;
   t1[3481] := 0.0189065;
   t1[3482] := 0.0200712;
   t1[3483] := 0.0206493;
   t1[3484] := 0.0207127;
   t1[3485] := 0.0203332;
   t1[3486] := 0.0195827;
   t1[3487] := 0.0185328;
   t1[3488] := 0.0172555;
   t1[3489] := 0.0158225;
   t1[3490] := 0.0143056;
   t1[3491] := 0.0127766;
   t1[3492] := 0.0113074;
   t1[3493] := 0.0099697;
   t1[3494] := 0.0088354;
   t1[3495] := 0.0079762;
   t1[3496] := 0.0074639;
   t1[3497] := 0.0073545;
   t1[3498] := 0.0076244;
   t1[3499] := 0.008225;
   t1[3500] := 0.0634489;
   t1[3501] := 0.0687754;
   t1[3502] := 0.0738956;
   t1[3503] := 0.0788046;
   t1[3504] := 0.0834973;
   t1[3505] := 0.0879686;
   t1[3506] := 0.0922134;
   t1[3507] := 0.0962268;
   t1[3508] := 0.1000032;
   t1[3509] := 0.1035297;
   t1[3510] := 0.1067877;
   t1[3511] := 0.1097582;
   t1[3512] := 0.1124226;
   t1[3513] := 0.1147619;
   t1[3514] := 0.1167574;
   t1[3515] := 0.1183902;
   t1[3516] := 0.1196415;
   t1[3517] := 0.1204924;
   t1[3518] := 0.1209241;
   t1[3519] := 0.1209178;
   t1[3520] := 0.1204547;
   t1[3521] := 0.1195159;
   t1[3522] := 0.1180827;
   t1[3523] := 0.1161361;
   t1[3524] := 0.1136574;
   t1[3525] := 0.1106277;
   t1[3526] := 0.1070282;
   t1[3527] := 0.1028402;
   t1[3528] := 0.098064;
   t1[3529] := 0.0927354;
   t1[3530] := 0.0868944;
   t1[3531] := 0.0805809;
   t1[3532] := 0.0738348;
   t1[3533] := 0.066696;
   t1[3534] := 0.0592045;
   t1[3535] := 0.0514001;
   t1[3536] := 0.0433228;
   t1[3537] := 0.0350125;
   t1[3538] := 0.0265092;
   t1[3539] := 0.0178526;
   t1[3540] := 0.0090829;
   t1[3541] := 0.0002397;
   t1[3542] := -0.0086368;
   t1[3543] := -0.0175068;
   t1[3544] := -0.0263304;
   t1[3545] := -0.0350677;
   t1[3546] := -0.0436787;
   t1[3547] := -0.0521247;
   t1[3548] := -0.0603729;
   t1[3549] := -0.0683924;
   t1[3550] := 0.1123488;
   t1[3551] := 0.1157331;
   t1[3552] := 0.1188747;
   t1[3553] := 0.1217489;
   t1[3554] := 0.1243309;
   t1[3555] := 0.1265962;
   t1[3556] := 0.1285198;
   t1[3557] := 0.1300773;
   t1[3558] := 0.1312449;
   t1[3559] := 0.1320146;
   t1[3560] := 0.1323908;
   t1[3561] := 0.1323781;
   t1[3562] := 0.1319812;
   t1[3563] := 0.1312049;
   t1[3564] := 0.1300538;
   t1[3565] := 0.1285327;
   t1[3566] := 0.1266461;
   t1[3567] := 0.1243988;
   t1[3568] := 0.1217955;
   t1[3569] := 0.1188409;
   t1[3570] := 0.1155397;
   t1[3571] := 0.1118965;
   t1[3572] := 0.107916;
   t1[3573] := 0.103603;
   t1[3574] := 0.0989621;
   t1[3575] := 0.093998;
   t1[3576] := 0.0887154;
   t1[3577] := 0.0831191;
   t1[3578] := 0.0772214;
   t1[3579] := 0.0710488;
   t1[3580] := 0.0646297;
   t1[3581] := 0.0579922;
   t1[3582] := 0.0511646;
   t1[3583] := 0.044175;
   t1[3584] := 0.0370518;
   t1[3585] := 0.0298231;
   t1[3586] := 0.0225172;
   t1[3587] := 0.0151622;
   t1[3588] := 0.0077865;
   t1[3589] := 0.0004181;
   t1[3590] := -0.0069146;
   t1[3591] := -0.0141834;
   t1[3592] := -0.0213601;
   t1[3593] := -0.0284165;
   t1[3594] := -0.0353244;
   t1[3595] := -0.0420555;
   t1[3596] := -0.0485816;
   t1[3597] := -0.054876;
   t1[3598] := -0.0609194;
   t1[3599] := -0.0666947;
   t1[3600] := 0.086788;
   t1[3601] := 0.0869916;
   t1[3602] := 0.0868084;
   t1[3603] := 0.0862098;
   t1[3604] := 0.0851675;
   t1[3605] := 0.0836532;
   t1[3606] := 0.0816382;
   t1[3607] := 0.0790944;
   t1[3608] := 0.0759956;
   t1[3609] := 0.0723527;
   t1[3610] := 0.0682055;
   t1[3611] := 0.0635948;
   t1[3612] := 0.058561;
   t1[3613] := 0.053145;
   t1[3614] := 0.0473873;
   t1[3615] := 0.0413286;
   t1[3616] := 0.0350095;
   t1[3617] := 0.0284707;
   t1[3618] := 0.0217528;
   t1[3619] := 0.0148965;
   t1[3620] := 0.0079425;
   t1[3621] := 0.0009313;
   t1[3622] := -0.0060964;
   t1[3623] := -0.0130999;
   t1[3624] := -0.0200386;
   t1[3625] := -0.0268718;
   t1[3626] := -0.0335589;
   t1[3627] := -0.0400593;
   t1[3628] := -0.0463343;
   t1[3629] := -0.0523494;
   t1[3630] := -0.0580704;
   t1[3631] := -0.063463;
   t1[3632] := -0.068493;
   t1[3633] := -0.0731262;
   t1[3634] := -0.0773285;
   t1[3635] := -0.0810656;
   t1[3636] := -0.0843032;
   t1[3637] := -0.0870073;
   t1[3638] := -0.0891435;
   t1[3639] := -0.0906777;
   t1[3640] := -0.0915757;
   t1[3641] := -0.0918033;
   t1[3642] := -0.0913262;
   t1[3643] := -0.0901102;
   t1[3644] := -0.0881213;
   t1[3645] := -0.085325;
   t1[3646] := -0.0816872;
   t1[3647] := -0.0771902;
   t1[3648] := -0.0718982;
   t1[3649] := -0.065901;
   t1[3650] := -0.2284766;
   t1[3651] := -0.2244241;
   t1[3652] := -0.2199992;
   t1[3653] := -0.2152239;
   t1[3654] := -0.2101205;
   t1[3655] := -0.2047109;
   t1[3656] := -0.1990172;
   t1[3657] := -0.1930615;
   t1[3658] := -0.1868655;
   t1[3659] := -0.1804436;
   t1[3660] := -0.1738047;
   t1[3661] := -0.1669575;
   t1[3662] := -0.1599106;
   t1[3663] := -0.1526729;
   t1[3664] := -0.1452529;
   t1[3665] := -0.1376594;
   t1[3666] := -0.1299012;
   t1[3667] := -0.1219868;
   t1[3668] := -0.1139251;
   t1[3669] := -0.1057247;
   t1[3670] := -0.0973943;
   t1[3671] := -0.0889426;
   t1[3672] := -0.0803784;
   t1[3673] := -0.0717103;
   t1[3674] := -0.062947;
   t1[3675] := -0.0540973;
   t1[3676] := -0.0451698;
   t1[3677] := -0.0361735;
   t1[3678] := -0.0271343;
   t1[3679] := -0.0181109;
   t1[3680] := -0.0091655;
   t1[3681] := -0.0003606;
   t1[3682] := 0.0082418;
   t1[3683] := 0.0165793;
   t1[3684] := 0.0245896;
   t1[3685] := 0.0322105;
   t1[3686] := 0.0393797;
   t1[3687] := 0.0460349;
   t1[3688] := 0.0521138;
   t1[3689] := 0.0575541;
   t1[3690] := 0.0622937;
   t1[3691] := 0.0662701;
   t1[3692] := 0.0694212;
   t1[3693] := 0.0716847;
   t1[3694] := 0.0729983;
   t1[3695] := 0.0732996;
   t1[3696] := 0.0725265;
   t1[3697] := 0.0706383;
   t1[3698] := 0.0677025;
   t1[3699] := 0.0638202;
   t1[3700] := 0.2277943;
   t1[3701] := 0.220762;
   t1[3702] := 0.2129452;
   t1[3703] := 0.2043566;
   t1[3704] := 0.1950092;
   t1[3705] := 0.1849158;
   t1[3706] := 0.1740893;
   t1[3707] := 0.1625425;
   t1[3708] := 0.1502897;
   t1[3709] := 0.1373665;
   t1[3710] := 0.1238251;
   t1[3711] := 0.1097184;
   t1[3712] := 0.0950992;
   t1[3713] := 0.0800201;
   t1[3714] := 0.0645341;
   t1[3715] := 0.0486939;
   t1[3716] := 0.0325522;
   t1[3717] := 0.0161619;
   t1[3718] := -0.0004242;
   t1[3719] := -0.0171534;
   t1[3720] := -0.0339729;
   t1[3721] := -0.0508299;
   t1[3722] := -0.0676715;
   t1[3723] := -0.0844452;
   t1[3724] := -0.1010979;
   t1[3725] := -0.117577;
   t1[3726] := -0.1338297;
   t1[3727] := -0.1498032;
   t1[3728] := -0.1654526;
   t1[3729] := -0.1807471;
   t1[3730] := -0.1956579;
   t1[3731] := -0.2101559;
   t1[3732] := -0.2242122;
   t1[3733] := -0.2377978;
   t1[3734] := -0.2508838;
   t1[3735] := -0.2634413;
   t1[3736] := -0.2754411;
   t1[3737] := -0.2868544;
   t1[3738] := -0.2976522;
   t1[3739] := -0.3078055;
   t1[3740] := -0.3172854;
   t1[3741] := -0.3260629;
   t1[3742] := -0.3341089;
   t1[3743] := -0.3413948;
   t1[3744] := -0.3478912;
   t1[3745] := -0.3535694;
   t1[3746] := -0.3584003;
   t1[3747] := -0.3623612;
   t1[3748] := -0.3654596;
   t1[3749] := -0.3677126;
